LIN {X 0,Y 361.829,Z 158.416,A -85,B 0,C 180,E1 -12912.828,E2 -12912.828} C_VEL
LIN {X 0,Y 361.81,Z 158.413,A -85,B 0,C 180,E1 -12915.946,E2 -12915.946} C_VEL
LIN {X 0,Y 361.807,Z 158.415,A -85,B 0,C 180,E1 -12919.248,E2 -12919.248} C_VEL
LIN {X 0,Y 361.859,Z 158.41,A -85,B 0,C 180,E1 -12922.98,E2 -12922.98} C_VEL
LIN {X 0,Y 361.853,Z 158.414,A -85,B 0,C 180,E1 -12926.63,E2 -12926.63} C_VEL
LIN {X 0,Y 361.85,Z 158.408,A -85,B 0,C 180,E1 -12929.669,E2 -12929.669} C_VEL
LIN {X 0,Y 361.849,Z 158.408,A -85,B 0,C 180,E1 -12933.466,E2 -12933.466} C_VEL
LIN {X 0,Y 361.855,Z 158.408,A -85,B 0,C 180,E1 -12937.142,E2 -12937.142} C_VEL
LIN {X 0,Y 361.851,Z 158.41,A -85,B 0,C 180,E1 -12940.72,E2 -12940.72} C_VEL
LIN {X 0,Y 361.888,Z 158.409,A -85,B 0,C 180,E1 -12944.223,E2 -12944.223} C_VEL
LIN {X 0,Y 361.992,Z 158.393,A -85,B 0,C 180,E1 -12946.527,E2 -12946.527} C_VEL
LIN {X 0,Y 361.987,Z 158.395,A -85,B 0,C 180,E1 -12949.936,E2 -12949.936} C_VEL
LIN {X 0,Y 362.114,Z 158.375,A -85,B 0,C 180,E1 -12953.312,E2 -12953.312} C_VEL
LIN {X 0,Y 362.256,Z 158.361,A -85,B 0,C 180,E1 -12957.776,E2 -12957.776} C_VEL
LIN {X 0,Y 362.166,Z 158.369,A -85,B 0,C 180,E1 -12961.112,E2 -12961.112} C_VEL
LIN {X 0,Y 362.256,Z 158.36,A -85,B 0,C 180,E1 -12962.223,E2 -12962.223} C_VEL
LIN {X 0,Y 362.113,Z 158.375,A -85,B 0,C 180,E1 -12966.687,E2 -12966.687} C_VEL
LIN {X 0,Y 361.987,Z 158.394,A -85,B 0,C 180,E1 -12970.063,E2 -12970.063} C_VEL
LIN {X 0,Y 361.972,Z 158.397,A -85,B 0,C 180,E1 -12973.887,E2 -12973.887} C_VEL
LIN {X 0,Y 361.876,Z 158.406,A -85,B 0,C 180,E1 -12978.103,E2 -12978.103} C_VEL
LIN {X 0,Y 361.845,Z 158.413,A -85,B 0,C 180,E1 -12981.656,E2 -12981.656} C_VEL
LIN {X 0,Y 361.852,Z 158.413,A -85,B 0,C 180,E1 -12985.296,E2 -12985.296} C_VEL
LIN {X 0,Y 361.848,Z 158.412,A -85,B 0,C 180,E1 -12989.074,E2 -12989.074} C_VEL
LIN {X 0,Y 361.84,Z 158.412,A -85,B 0,C 180,E1 -12992.946,E2 -12992.946} C_VEL
LIN {X 0,Y 361.857,Z 158.409,A -85,B 0,C 180,E1 -12995.638,E2 -12995.638} C_VEL
LIN {X 0,Y 361.819,Z 158.417,A -85,B 0,C 180,E1 -12999.018,E2 -12999.018} C_VEL
LIN {X 0,Y 361.823,Z 158.415,A -85,B 0,C 180,E1 -13002.831,E2 -13002.831} C_VEL
LIN {X 0,Y 361.808,Z 158.413,A -85,B 0,C 180,E1 -13005.948,E2 -13005.948} C_VEL
LIN {X 0,Y 361.805,Z 158.416,A -85,B 0,C 180,E1 -13009.25,E2 -13009.25} C_VEL
LIN {X 0,Y 361.856,Z 158.412,A -85,B 0,C 180,E1 -13012.982,E2 -13012.982} C_VEL
LIN {X 0,Y 361.853,Z 158.412,A -85,B 0,C 180,E1 -13016.632,E2 -13016.632} C_VEL
LIN {X 0,Y 361.844,Z 158.411,A -85,B 0,C 180,E1 -13019.671,E2 -13019.671} C_VEL
LIN {X 0,Y 361.862,Z 158.495,A -85,B 0,C 180,E1 -13021.035,E2 -13021.035} C_VEL
LIN {X 0,Y 364.381,Z 171.266,A -85,B 0,C 180,E1 -13024.282,E2 -13024.282} C_VEL
LIN {X 0,Y 365.151,Z 176.441,A -85,B 0,C 180,E1 -13025.557,E2 -13025.557} C_VEL
LIN {X 0,Y 364.358,Z 186.129,A -85,B 0,C 180,E1 -13027.799,E2 -13027.799} C_VEL
LIN {X 0,Y 363.991,Z 190.26,A -85,B 0,C 180,E1 -13028.747,E2 -13028.747} C_VEL
LIN {X 0,Y 368.452,Z 222.561,A -85,B 0,C 180,E1 -13029.729,E2 -13029.729} C_VEL
LIN {X 0,Y 366.841,Z 299.767,A -85,B 0,C 180,E1 -13031.501,E2 -13031.501} C_VEL
LIN {X 0,Y 366.187,Z 313.467,A -85,B 0,C 180,E1 -13032.046,E2 -13032.046} C_VEL
LIN {X 0,Y 365.37,Z 326.351,A -85,B 0,C 180,E1 -13032.799,E2 -13032.799} C_VEL
LIN {X 0,Y 364.524,Z 338.673,A -85,B 0,C 180,E1 -13033.767,E2 -13033.767} C_VEL
LIN {X 0,Y 363.673,Z 349.679,A -85,B 0,C 180,E1 -13034.87,E2 -13034.87} C_VEL
LIN {X 0,Y 362.818,Z 360.759,A -85,B 0,C 180,E1 -13036.274,E2 -13036.274} C_VEL
LIN {X 0,Y 362.039,Z 369.703,A -85,B 0,C 180,E1 -13037.671,E2 -13037.671} C_VEL
LIN {X 0,Y 361.369,Z 377.07,A -85,B 0,C 180,E1 -13039.07,E2 -13039.07} C_VEL
LIN {X 0,Y 360.899,Z 384.28,A -85,B 0,C 180,E1 -13040.756,E2 -13040.756} C_VEL
LIN {X 0,Y 360.584,Z 390.846,A -85,B 0,C 180,E1 -13042.723,E2 -13042.723} C_VEL
LIN {X 0,Y 360.382,Z 395.127,A -85,B 0,C 180,E1 -13044.405,E2 -13044.405} C_VEL
LIN {X 0,Y 360.386,Z 397.376,A -85,B 0,C 180,E1 -13045.527,E2 -13045.527} C_VEL
LIN {X 0,Y 360.304,Z 399.111,A -85,B 0,C 180,E1 -13046.646,E2 -13046.646} C_VEL
LIN {X 0,Y 360.279,Z 400.423,A -85,B 0,C 180,E1 -13047.765,E2 -13047.765} C_VEL
LIN {X 0,Y 360.322,Z 401.322,A -85,B 0,C 180,E1 -13048.883,E2 -13048.883} C_VEL
LIN {X 0,Y 360.36,Z 401.765,A -85,B 0,C 180,E1 -13050.001,E2 -13050.001} C_VEL
LIN {X 0,Y 360.303,Z 401.777,A -85,B 0,C 180,E1 -13051.119,E2 -13051.119} C_VEL
LIN {X 0,Y 360.262,Z 401.385,A -85,B 0,C 180,E1 -13052.237,E2 -13052.237} C_VEL
LIN {X 0,Y 360.296,Z 400.589,A -85,B 0,C 180,E1 -13053.356,E2 -13053.356} C_VEL
LIN {X 0,Y 360.346,Z 399.333,A -85,B 0,C 180,E1 -13054.475,E2 -13054.475} C_VEL
LIN {X 0,Y 360.378,Z 397.037,A -85,B 0,C 180,E1 -13055.962,E2 -13055.962} C_VEL
LIN {X 0,Y 360.695,Z 392.947,A -85,B 0,C 180,E1 -13057.84,E2 -13057.84} C_VEL
LIN {X 0,Y 361.149,Z 388.099,A -85,B 0,C 180,E1 -13059.522,E2 -13059.522} C_VEL
LIN {X 0,Y 361.921,Z 380.826,A -85,B 0,C 180,E1 -13061.482,E2 -13061.482} C_VEL
LIN {X 0,Y 362.96,Z 372.947,A -85,B 0,C 180,E1 -13063.152,E2 -13063.152} C_VEL
LIN {X 0,Y 364.128,Z 363.132,A -85,B 0,C 180,E1 -13064.812,E2 -13064.812} C_VEL
LIN {X 0,Y 365.247,Z 353.009,A -85,B 0,C 180,E1 -13066.202,E2 -13066.202} C_VEL
LIN {X 0,Y 366.61,Z 341.672,A -85,B 0,C 180,E1 -13067.431,E2 -13067.431} C_VEL
LIN {X 0,Y 367.795,Z 330.68,A -85,B 0,C 180,E1 -13068.379,E2 -13068.379} C_VEL
LIN {X 0,Y 368.792,Z 318.696,A -85,B 0,C 180,E1 -13069.193,E2 -13069.193} C_VEL
LIN {X 0,Y 369.825,Z 305.614,A -85,B 0,C 180,E1 -13069.823,E2 -13069.823} C_VEL
LIN {X 0,Y 370.495,Z 292.075,A -85,B 0,C 180,E1 -13070.255,E2 -13070.255} C_VEL
LIN {X 0,Y 372.443,Z 222.981,A -85,B 0,C 180,E1 -13071.896,E2 -13071.896} C_VEL
LIN {X 0,Y 369.403,Z 203.708,A -85,B 0,C 180,E1 -13072.672,E2 -13072.672} C_VEL
LIN {X 0,Y 365.96,Z 188.136,A -85,B 0,C 180,E1 -13073.424,E2 -13073.424} C_VEL
LIN {X 0,Y 366.691,Z 181.612,A -85,B 0,C 180,E1 -13074.94,E2 -13074.94} C_VEL
LIN {X 0,Y 366.084,Z 176.728,A -85,B 0,C 180,E1 -13076.204,E2 -13076.204} C_VEL
LIN {X 0,Y 364.044,Z 167.054,A -85,B 0,C 180,E1 -13078.859,E2 -13078.859} C_VEL
LIN {X 0,Y 361.855,Z 158.412,A -85,B 0,C 180,E1 -13081.462,E2 -13081.462} C_VEL
LIN {X 0,Y 361.853,Z 158.411,A -85,B 0,C 180,E1 -13084.281,E2 -13084.281} C_VEL
LIN {X 0,Y 361.86,Z 158.409,A -85,B 0,C 180,E1 -13087.222,E2 -13087.222} C_VEL
LIN {X 0,Y 361.814,Z 158.417,A -85,B 0,C 180,E1 -13090.751,E2 -13090.751} C_VEL
LIN {X 0,Y 361.815,Z 158.413,A -85,B 0,C 180,E1 -13094.37,E2 -13094.37} C_VEL
LIN {X 0,Y 361.832,Z 158.409,A -85,B 0,C 180,E1 -13097.57,E2 -13097.57} C_VEL
LIN {X 0,Y 361.845,Z 158.405,A -85,B 0,C 180,E1 -13101.572,E2 -13101.572} C_VEL
LIN {X 0,Y 361.873,Z 158.407,A -85,B 0,C 180,E1 -13104.657,E2 -13104.657} C_VEL
LIN {X 0,Y 361.841,Z 158.413,A -85,B 0,C 180,E1 -13108.371,E2 -13108.371} C_VEL
LIN {X 0,Y 361.87,Z 158.406,A -85,B 0,C 180,E1 -13110.953,E2 -13110.953} C_VEL
LIN {X 0,Y 361.869,Z 158.405,A -85,B 0,C 180,E1 -13114.706,E2 -13114.706} C_VEL
LIN {X 0,Y 361.858,Z 158.41,A -85,B 0,C 180,E1 -13118.345,E2 -13118.345} C_VEL
LIN {X 0,Y 361.908,Z 158.403,A -85,B 0,C 180,E1 -13122.093,E2 -13122.093} C_VEL
LIN {X 0,Y 361.984,Z 158.394,A -85,B 0,C 180,E1 -13126.114,E2 -13126.114} C_VEL
LIN {X 0,Y 362.004,Z 158.394,A -85,B 0,C 180,E1 -13129.937,E2 -13129.937} C_VEL
LIN {X 0,Y 362.126,Z 158.38,A -85,B 0,C 180,E1 -13133.313,E2 -13133.313} C_VEL
LIN {X 0,Y 362.269,Z 158.361,A -85,B 0,C 180,E1 -13137.777,E2 -13137.777} C_VEL
LIN {X 0,Y 362.185,Z 158.387,A -85,B 0,C 180,E1 -13140.556,E2 -13140.556} C_VEL
LIN {X 0,Y 363.973,Z 165.762,A -85,B 0,C 180,E1 -13142.767,E2 -13142.767} C_VEL
LIN {X 0,Y 365.318,Z 172.142,A -85,B 0,C 180,E1 -13144.584,E2 -13144.584} C_VEL
LIN {X 0,Y 369.751,Z 182.829,A -85,B 0,C 180,E1 -13145.285,E2 -13145.285} C_VEL
LIN {X 0,Y 373.135,Z 198.483,A -85,B 0,C 180,E1 -13146,E2 -13146} C_VEL
LIN {X 0,Y 370.496,Z 280.618,A -85,B 0,C 180,E1 -13147.976,E2 -13147.976} C_VEL
LIN {X 0,Y 369.775,Z 293.95,A -85,B 0,C 180,E1 -13148.511,E2 -13148.511} C_VEL
LIN {X 0,Y 368.967,Z 305.625,A -85,B 0,C 180,E1 -13149.18,E2 -13149.18} C_VEL
LIN {X 0,Y 368.052,Z 316.889,A -85,B 0,C 180,E1 -13150.035,E2 -13150.035} C_VEL
LIN {X 0,Y 366.76,Z 329.226,A -85,B 0,C 180,E1 -13151.235,E2 -13151.235} C_VEL
LIN {X 0,Y 365.557,Z 339.475,A -85,B 0,C 180,E1 -13152.491,E2 -13152.491} C_VEL
LIN {X 0,Y 364.345,Z 349.032,A -85,B 0,C 180,E1 -13153.953,E2 -13153.953} C_VEL
LIN {X 0,Y 363.334,Z 357.164,A -85,B 0,C 180,E1 -13155.481,E2 -13155.481} C_VEL
LIN {X 0,Y 362.367,Z 364.439,A -85,B 0,C 180,E1 -13157.168,E2 -13157.168} C_VEL
LIN {X 0,Y 361.68,Z 369.722,A -85,B 0,C 180,E1 -13158.701,E2 -13158.701} C_VEL
LIN {X 0,Y 361.113,Z 374.595,A -85,B 0,C 180,E1 -13160.507,E2 -13160.507} C_VEL
LIN {X 0,Y 360.705,Z 378.217,A -85,B 0,C 180,E1 -13162.33,E2 -13162.33} C_VEL
LIN {X 0,Y 360.373,Z 380.677,A -85,B 0,C 180,E1 -13164.177,E2 -13164.177} C_VEL
LIN {X 0,Y 360.186,Z 382.039,A -85,B 0,C 180,E1 -13166.159,E2 -13166.159} C_VEL
LIN {X 0,Y 360.109,Z 381.931,A -85,B 0,C 180,E1 -13168.569,E2 -13168.569} C_VEL
LIN {X 0,Y 360.203,Z 380.066,A -85,B 0,C 180,E1 -13170.851,E2 -13170.851} C_VEL
LIN {X 0,Y 360.384,Z 377.741,A -85,B 0,C 180,E1 -13172.404,E2 -13172.404} C_VEL
LIN {X 0,Y 360.626,Z 373.429,A -85,B 0,C 180,E1 -13174.414,E2 -13174.414} C_VEL
LIN {X 0,Y 361.062,Z 367.492,A -85,B 0,C 180,E1 -13176.413,E2 -13176.413} C_VEL
LIN {X 0,Y 361.561,Z 361.004,A -85,B 0,C 180,E1 -13178.109,E2 -13178.109} C_VEL
LIN {X 0,Y 362.205,Z 352.769,A -85,B 0,C 180,E1 -13179.816,E2 -13179.816} C_VEL
LIN {X 0,Y 362.997,Z 343.553,A -85,B 0,C 180,E1 -13181.354,E2 -13181.354} C_VEL
LIN {X 0,Y 363.79,Z 333.043,A -85,B 0,C 180,E1 -13182.766,E2 -13182.766} C_VEL
LIN {X 0,Y 364.669,Z 322.16,A -85,B 0,C 180,E1 -13183.933,E2 -13183.933} C_VEL
LIN {X 0,Y 365.522,Z 310.748,A -85,B 0,C 180,E1 -13184.906,E2 -13184.906} C_VEL
LIN {X 0,Y 366.232,Z 298.142,A -85,B 0,C 180,E1 -13185.728,E2 -13185.728} C_VEL
LIN {X 0,Y 366.765,Z 284.578,A -85,B 0,C 180,E1 -13186.361,E2 -13186.361} C_VEL
LIN {X 0,Y 367.225,Z 270.752,A -85,B 0,C 180,E1 -13186.757,E2 -13186.757} C_VEL
LIN {X 0,Y 368.691,Z 195.693,A -85,B 0,C 180,E1 -13188.451,E2 -13188.451} C_VEL
LIN {X 0,Y 364.189,Z 170.992,A -85,B 0,C 180,E1 -13189.268,E2 -13189.268} C_VEL
LIN {X 0,Y 362.217,Z 160.038,A -85,B 0,C 180,E1 -13192.264,E2 -13192.264} C_VEL
LIN {X 0,Y 361.902,Z 158.407,A -85,B 0,C 180,E1 -13192.77,E2 -13192.77} C_VEL
LIN {X 0,Y 361.859,Z 158.407,A -85,B 0,C 180,E1 -13195.719,E2 -13195.719} C_VEL
LIN {X 0,Y 361.852,Z 158.408,A -85,B 0,C 180,E1 -13199.669,E2 -13199.669} C_VEL
LIN {X 0,Y 361.859,Z 158.407,A -85,B 0,C 180,E1 -13203.467,E2 -13203.467} C_VEL
LIN {X 0,Y 361.866,Z 158.406,A -85,B 0,C 180,E1 -13207.142,E2 -13207.142} C_VEL
LIN {X 0,Y 361.848,Z 158.41,A -85,B 0,C 180,E1 -13210.719,E2 -13210.719} C_VEL
LIN {X 0,Y 361.882,Z 158.404,A -85,B 0,C 180,E1 -13213.063,E2 -13213.063} C_VEL
LIN {X 0,Y 362.004,Z 158.391,A -85,B 0,C 180,E1 -13216.527,E2 -13216.527} C_VEL
LIN {X 0,Y 362,Z 158.395,A -85,B 0,C 180,E1 -13219.936,E2 -13219.936} C_VEL
LIN {X 0,Y 362.123,Z 158.375,A -85,B 0,C 180,E1 -13223.312,E2 -13223.312} C_VEL
LIN {X 0,Y 362.268,Z 158.361,A -85,B 0,C 180,E1 -13227.775,E2 -13227.775} C_VEL
LIN {X 0,Y 362.177,Z 158.368,A -85,B 0,C 180,E1 -13231.111,E2 -13231.111} C_VEL
LIN {X 0,Y 362.268,Z 158.358,A -85,B 0,C 180,E1 -13232.223,E2 -13232.223} C_VEL
LIN {X 0,Y 362.121,Z 158.374,A -85,B 0,C 180,E1 -13236.686,E2 -13236.686} C_VEL
LIN {X 0,Y 361.998,Z 158.391,A -85,B 0,C 180,E1 -13240.062,E2 -13240.062} C_VEL
LIN {X 0,Y 361.945,Z 158.395,A -85,B 0,C 180,E1 -13242.003,E2 -13242.003} C_VEL
LIN {X 0,Y 361.283,Z 158.481,A -85,B 0,C 180,E1 -13242.931,E2 -13242.931} C_VEL
LIN {X 0,Y 358.386,Z 158.839,A -85,B 0,C 180,E1 -13244.441,E2 -13244.441} C_VEL
LIN {X 0,Y 355.935,Z 159.149,A -85,B 0,C 180,E1 -13245.662,E2 -13245.662} C_VEL
LIN {X 0,Y 354.901,Z 159.274,A -85,B 0,C 180,E1 -13246.608,E2 -13246.608} C_VEL
LIN {X 0,Y 354.827,Z 159.284,A -85,B 0,C 180,E1 -13246.928,E2 -13246.928} C_VEL
LIN {X 0,Y 354.79,Z 159.291,A -85,B 0,C 180,E1 -13249.678,E2 -13249.678} C_VEL
LIN {X 0,Y 354.806,Z 159.286,A -85,B 0,C 180,E1 -13252.107,E2 -13252.107} C_VEL
LIN {X 0,Y 354.799,Z 159.287,A -85,B 0,C 180,E1 -13255.834,E2 -13255.834} C_VEL
LIN {X 0,Y 354.792,Z 159.289,A -85,B 0,C 180,E1 -13259.683,E2 -13259.683} C_VEL
LIN {X 0,Y 354.785,Z 159.288,A -85,B 0,C 180,E1 -13262.332,E2 -13262.332} C_VEL
LIN {X 0,Y 354.817,Z 159.285,A -85,B 0,C 180,E1 -13265.697,E2 -13265.697} C_VEL
LIN {X 0,Y 354.766,Z 159.293,A -85,B 0,C 180,E1 -13269.411,E2 -13269.411} C_VEL
LIN {X 0,Y 354.781,Z 159.294,A -85,B 0,C 180,E1 -13272.865,E2 -13272.865} C_VEL
LIN {X 0,Y 354.759,Z 159.292,A -85,B 0,C 180,E1 -13276.102,E2 -13276.102} C_VEL
LIN {X 0,Y 354.76,Z 159.294,A -85,B 0,C 180,E1 -13279.175,E2 -13279.175} C_VEL
LIN {X 0,Y 354.796,Z 159.29,A -85,B 0,C 180,E1 -13282.403,E2 -13282.403} C_VEL
LIN {X 0,Y 354.806,Z 159.289,A -85,B 0,C 180,E1 -13284.94,E2 -13284.94} C_VEL
LIN {X 0,Y 354.788,Z 159.292,A -85,B 0,C 180,E1 -13288.404,E2 -13288.404} C_VEL
LIN {X 0,Y 354.791,Z 159.287,A -85,B 0,C 180,E1 -13291.613,E2 -13291.613} C_VEL
LIN {X 0,Y 354.795,Z 159.287,A -85,B 0,C 180,E1 -13295.418,E2 -13295.418} C_VEL
LIN {X 0,Y 354.815,Z 159.285,A -85,B 0,C 180,E1 -13299.112,E2 -13299.112} C_VEL
LIN {X 0,Y 354.845,Z 159.283,A -85,B 0,C 180,E1 -13302.717,E2 -13302.717} C_VEL
LIN {X 0,Y 354.932,Z 159.276,A -85,B 0,C 180,E1 -13306.254,E2 -13306.254} C_VEL
LIN {X 0,Y 354.944,Z 159.27,A -85,B 0,C 180,E1 -13309.735,E2 -13309.735} C_VEL
LIN {X 0,Y 355.08,Z 159.251,A -85,B 0,C 180,E1 -13313.179,E2 -13313.179} C_VEL
LIN {X 0,Y 355.218,Z 159.238,A -85,B 0,C 180,E1 -13317.732,E2 -13317.732} C_VEL
LIN {X 0,Y 355.137,Z 159.244,A -85,B 0,C 180,E1 -13321.134,E2 -13321.134} C_VEL
LIN {X 0,Y 355.218,Z 159.237,A -85,B 0,C 180,E1 -13322.268,E2 -13322.268} C_VEL
LIN {X 0,Y 355.079,Z 159.251,A -85,B 0,C 180,E1 -13326.82,E2 -13326.82} C_VEL
LIN {X 0,Y 354.943,Z 159.27,A -85,B 0,C 180,E1 -13330.265,E2 -13330.265} C_VEL
LIN {X 0,Y 354.915,Z 159.274,A -85,B 0,C 180,E1 -13334.005,E2 -13334.005} C_VEL
LIN {X 0,Y 354.834,Z 159.284,A -85,B 0,C 180,E1 -13338.068,E2 -13338.068} C_VEL
LIN {X 0,Y 354.798,Z 159.287,A -85,B 0,C 180,E1 -13342.108,E2 -13342.108} C_VEL
LIN {X 0,Y 354.791,Z 159.289,A -85,B 0,C 180,E1 -13345.836,E2 -13345.836} C_VEL
LIN {X 0,Y 354.786,Z 159.291,A -85,B 0,C 180,E1 -13349.685,E2 -13349.685} C_VEL
LIN {X 0,Y 354.779,Z 159.289,A -85,B 0,C 180,E1 -13352.334,E2 -13352.334} C_VEL
LIN {X 0,Y 354.811,Z 159.286,A -85,B 0,C 180,E1 -13355.699,E2 -13355.699} C_VEL
LIN {X 0,Y 354.762,Z 159.294,A -85,B 0,C 180,E1 -13359.413,E2 -13359.413} C_VEL
LIN {X 0,Y 354.775,Z 159.294,A -85,B 0,C 180,E1 -13362.867,E2 -13362.867} C_VEL
LIN {X 0,Y 354.757,Z 159.292,A -85,B 0,C 180,E1 -13366.104,E2 -13366.104} C_VEL
LIN {X 0,Y 354.758,Z 159.295,A -85,B 0,C 180,E1 -13369.176,E2 -13369.176} C_VEL
LIN {X 0,Y 354.794,Z 159.289,A -85,B 0,C 180,E1 -13372.405,E2 -13372.405} C_VEL
LIN {X 0,Y 354.804,Z 159.29,A -85,B 0,C 180,E1 -13374.941,E2 -13374.941} C_VEL
LIN {X 0,Y 354.789,Z 159.29,A -85,B 0,C 180,E1 -13378.406,E2 -13378.406} C_VEL
LIN {X 0,Y 354.835,Z 159.397,A -85,B 0,C 180,E1 -13380.785,E2 -13380.785} C_VEL
LIN {X 0,Y 357.303,Z 171.951,A -85,B 0,C 180,E1 -13384.047,E2 -13384.047} C_VEL
LIN {X 0,Y 358.162,Z 177.252,A -85,B 0,C 180,E1 -13385.381,E2 -13385.381} C_VEL
LIN {X 0,Y 357.441,Z 186.368,A -85,B 0,C 180,E1 -13387.535,E2 -13387.535} C_VEL
LIN {X 0,Y 357.061,Z 190.013,A -85,B 0,C 180,E1 -13388.388,E2 -13388.388} C_VEL
LIN {X 0,Y 361.633,Z 222.954,A -85,B 0,C 180,E1 -13389.432,E2 -13389.432} C_VEL
LIN {X 0,Y 360.006,Z 298.965,A -85,B 0,C 180,E1 -13391.21,E2 -13391.21} C_VEL
LIN {X 0,Y 359.316,Z 312.831,A -85,B 0,C 180,E1 -13391.764,E2 -13391.764} C_VEL
LIN {X 0,Y 358.554,Z 324.868,A -85,B 0,C 180,E1 -13392.462,E2 -13392.462} C_VEL
LIN {X 0,Y 357.658,Z 337.442,A -85,B 0,C 180,E1 -13393.447,E2 -13393.447} C_VEL
LIN {X 0,Y 356.733,Z 348.739,A -85,B 0,C 180,E1 -13394.577,E2 -13394.577} C_VEL
LIN {X 0,Y 355.978,Z 358.93,A -85,B 0,C 180,E1 -13395.86,E2 -13395.86} C_VEL
LIN {X 0,Y 355.079,Z 368.978,A -85,B 0,C 180,E1 -13397.426,E2 -13397.426} C_VEL
LIN {X 0,Y 354.35,Z 376.436,A -85,B 0,C 180,E1 -13398.851,E2 -13398.851} C_VEL
LIN {X 0,Y 353.851,Z 383.761,A -85,B 0,C 180,E1 -13400.57,E2 -13400.57} C_VEL
LIN {X 0,Y 353.57,Z 388.695,A -85,B 0,C 180,E1 -13402.003,E2 -13402.003} C_VEL
LIN {X 0,Y 353.313,Z 394.163,A -85,B 0,C 180,E1 -13404.036,E2 -13404.036} C_VEL
LIN {X 0,Y 353.297,Z 397.027,A -85,B 0,C 180,E1 -13405.437,E2 -13405.437} C_VEL
LIN {X 0,Y 353.227,Z 398.801,A -85,B 0,C 180,E1 -13406.579,E2 -13406.579} C_VEL
LIN {X 0,Y 353.186,Z 400.136,A -85,B 0,C 180,E1 -13407.72,E2 -13407.72} C_VEL
LIN {X 0,Y 353.223,Z 401.059,A -85,B 0,C 180,E1 -13408.861,E2 -13408.861} C_VEL
LIN {X 0,Y 353.263,Z 401.552,A -85,B 0,C 180,E1 -13410.001,E2 -13410.001} C_VEL
LIN {X 0,Y 353.203,Z 401.589,A -85,B 0,C 180,E1 -13411.141,E2 -13411.141} C_VEL
LIN {X 0,Y 353.17,Z 401.223,A -85,B 0,C 180,E1 -13412.282,E2 -13412.282} C_VEL
LIN {X 0,Y 353.217,Z 400.456,A -85,B 0,C 180,E1 -13413.423,E2 -13413.423} C_VEL
LIN {X 0,Y 353.259,Z 399.246,A -85,B 0,C 180,E1 -13414.565,E2 -13414.565} C_VEL
LIN {X 0,Y 353.276,Z 397.264,A -85,B 0,C 180,E1 -13415.906,E2 -13415.906} C_VEL
LIN {X 0,Y 353.661,Z 392.957,A -85,B 0,C 180,E1 -13417.997,E2 -13417.997} C_VEL
LIN {X 0,Y 354.115,Z 388.159,A -85,B 0,C 180,E1 -13419.713,E2 -13419.713} C_VEL
LIN {X 0,Y 354.95,Z 380.941,A -85,B 0,C 180,E1 -13421.71,E2 -13421.71} C_VEL
LIN {X 0,Y 356.051,Z 373.182,A -85,B 0,C 180,E1 -13423.412,E2 -13423.412} C_VEL
LIN {X 0,Y 357.243,Z 363.769,A -85,B 0,C 180,E1 -13425.063,E2 -13425.063} C_VEL
LIN {X 0,Y 358.315,Z 354.591,A -85,B 0,C 180,E1 -13426.378,E2 -13426.378} C_VEL
LIN {X 0,Y 359.744,Z 343.77,A -85,B 0,C 180,E1 -13427.627,E2 -13427.627} C_VEL
LIN {X 0,Y 361.11,Z 331.597,A -85,B 0,C 180,E1 -13428.732,E2 -13428.732} C_VEL
LIN {X 0,Y 362.247,Z 318.821,A -85,B 0,C 180,E1 -13429.627,E2 -13429.627} C_VEL
LIN {X 0,Y 363.347,Z 305.934,A -85,B 0,C 180,E1 -13430.265,E2 -13430.265} C_VEL
LIN {X 0,Y 364.059,Z 291.534,A -85,B 0,C 180,E1 -13430.74,E2 -13430.74} C_VEL
LIN {X 0,Y 366.159,Z 223.616,A -85,B 0,C 180,E1 -13432.4,E2 -13432.4} C_VEL
LIN {X 0,Y 362.975,Z 203.973,A -85,B 0,C 180,E1 -13433.224,E2 -13433.224} C_VEL
LIN {X 0,Y 359.419,Z 187.839,A -85,B 0,C 180,E1 -13434.053,E2 -13434.053} C_VEL
LIN {X 0,Y 359.866,Z 182.107,A -85,B 0,C 180,E1 -13435.446,E2 -13435.446} C_VEL
LIN {X 0,Y 358.089,Z 172.427,A -85,B 0,C 180,E1 -13438.102,E2 -13438.102} C_VEL
LIN {X 0,Y 355.787,Z 162.976,A -85,B 0,C 180,E1 -13440.904,E2 -13440.904} C_VEL
LIN {X 0,Y 354.776,Z 159.295,A -85,B 0,C 180,E1 -13442.125,E2 -13442.125} C_VEL
LIN {X 0,Y 354.821,Z 159.286,A -85,B 0,C 180,E1 -13445.699,E2 -13445.699} C_VEL
LIN {X 0,Y 354.771,Z 159.295,A -85,B 0,C 180,E1 -13449.413,E2 -13449.413} C_VEL
LIN {X 0,Y 354.785,Z 159.29,A -85,B 0,C 180,E1 -13452.867,E2 -13452.867} C_VEL
LIN {X 0,Y 354.766,Z 159.286,A -85,B 0,C 180,E1 -13456.103,E2 -13456.103} C_VEL
LIN {X 0,Y 354.768,Z 159.287,A -85,B 0,C 180,E1 -13459.176,E2 -13459.176} C_VEL
LIN {X 0,Y 354.802,Z 159.287,A -85,B 0,C 180,E1 -13462.405,E2 -13462.405} C_VEL
LIN {X 0,Y 354.812,Z 159.29,A -85,B 0,C 180,E1 -13464.941,E2 -13464.941} C_VEL
LIN {X 0,Y 354.797,Z 159.289,A -85,B 0,C 180,E1 -13468.406,E2 -13468.406} C_VEL
LIN {X 0,Y 354.8,Z 159.285,A -85,B 0,C 180,E1 -13471.615,E2 -13471.615} C_VEL
LIN {X 0,Y 354.809,Z 159.286,A -85,B 0,C 180,E1 -13475.42,E2 -13475.42} C_VEL
LIN {X 0,Y 354.828,Z 159.28,A -85,B 0,C 180,E1 -13479.113,E2 -13479.113} C_VEL
LIN {X 0,Y 354.856,Z 159.283,A -85,B 0,C 180,E1 -13482.718,E2 -13482.718} C_VEL
LIN {X 0,Y 354.944,Z 159.271,A -85,B 0,C 180,E1 -13486.255,E2 -13486.255} C_VEL
LIN {X 0,Y 354.96,Z 159.272,A -85,B 0,C 180,E1 -13489.736,E2 -13489.736} C_VEL
LIN {X 0,Y 355.092,Z 159.256,A -85,B 0,C 180,E1 -13493.18,E2 -13493.18} C_VEL
LIN {X 0,Y 355.231,Z 159.237,A -85,B 0,C 180,E1 -13497.733,E2 -13497.733} C_VEL
LIN {X 0,Y 355.177,Z 159.338,A -85,B 0,C 180,E1 -13499.929,E2 -13499.929} C_VEL
LIN {X 0,Y 357.062,Z 166.798,A -85,B 0,C 180,E1 -13502.256,E2 -13502.256} C_VEL
LIN {X 0,Y 358.228,Z 172.673,A -85,B 0,C 180,E1 -13503.913,E2 -13503.913} C_VEL
LIN {X 0,Y 363.645,Z 184.715,A -85,B 0,C 180,E1 -13504.79,E2 -13504.79} C_VEL
LIN {X 0,Y 366.878,Z 199.629,A -85,B 0,C 180,E1 -13505.497,E2 -13505.497} C_VEL
LIN {X 0,Y 364.075,Z 281.33,A -85,B 0,C 180,E1 -13507.522,E2 -13507.522} C_VEL
LIN {X 0,Y 363.327,Z 294.218,A -85,B 0,C 180,E1 -13508.055,E2 -13508.055} C_VEL
LIN {X 0,Y 362.4,Z 306.756,A -85,B 0,C 180,E1 -13508.797,E2 -13508.797} C_VEL
LIN {X 0,Y 361.251,Z 319.341,A -85,B 0,C 180,E1 -13509.801,E2 -13509.801} C_VEL
LIN {X 0,Y 359.999,Z 330.799,A -85,B 0,C 180,E1 -13510.973,E2 -13510.973} C_VEL
LIN {X 0,Y 358.695,Z 340.853,A -85,B 0,C 180,E1 -13512.264,E2 -13512.264} C_VEL
LIN {X 0,Y 357.529,Z 349.603,A -85,B 0,C 180,E1 -13513.644,E2 -13513.644} C_VEL
LIN {X 0,Y 356.483,Z 357.482,A -85,B 0,C 180,E1 -13515.164,E2 -13515.164} C_VEL
LIN {X 0,Y 355.426,Z 364.981,A -85,B 0,C 180,E1 -13516.958,E2 -13516.958} C_VEL
LIN {X 0,Y 354.715,Z 370.084,A -85,B 0,C 180,E1 -13518.483,E2 -13518.483} C_VEL
LIN {X 0,Y 354.098,Z 374.921,A -85,B 0,C 180,E1 -13520.325,E2 -13520.325} C_VEL
LIN {X 0,Y 353.661,Z 378.511,A -85,B 0,C 180,E1 -13522.184,E2 -13522.184} C_VEL
LIN {X 0,Y 353.35,Z 380.682,A -85,B 0,C 180,E1 -13523.803,E2 -13523.803} C_VEL
LIN {X 0,Y 353.093,Z 382.221,A -85,B 0,C 180,E1 -13525.97,E2 -13525.97} C_VEL
LIN {X 0,Y 353.003,Z 382.453,A -85,B 0,C 180,E1 -13527.253,E2 -13527.253} C_VEL
LIN {X 0,Y 353.014,Z 381.969,A -85,B 0,C 180,E1 -13528.838,E2 -13528.838} C_VEL
LIN {X 0,Y 353.032,Z 381.26,A -85,B 0,C 180,E1 -13529.848,E2 -13529.848} C_VEL
LIN {X 0,Y 353.185,Z 378.877,A -85,B 0,C 180,E1 -13531.825,E2 -13531.825} C_VEL
LIN {X 0,Y 353.48,Z 375.079,A -85,B 0,C 180,E1 -13533.829,E2 -13533.829} C_VEL
LIN {X 0,Y 353.704,Z 370.93,A -85,B 0,C 180,E1 -13535.445,E2 -13535.445} C_VEL
LIN {X 0,Y 354.123,Z 365.839,A -85,B 0,C 180,E1 -13537.017,E2 -13537.017} C_VEL
LIN {X 0,Y 354.651,Z 359.392,A -85,B 0,C 180,E1 -13538.626,E2 -13538.626} C_VEL
LIN {X 0,Y 355.391,Z 350.69,A -85,B 0,C 180,E1 -13540.377,E2 -13540.377} C_VEL
LIN {X 0,Y 356.164,Z 341.093,A -85,B 0,C 180,E1 -13541.915,E2 -13541.915} C_VEL
LIN {X 0,Y 357.106,Z 330.02,A -85,B 0,C 180,E1 -13543.342,E2 -13543.342} C_VEL
LIN {X 0,Y 357.916,Z 319.863,A -85,B 0,C 180,E1 -13544.39,E2 -13544.39} C_VEL
LIN {X 0,Y 358.774,Z 308.064,A -85,B 0,C 180,E1 -13545.353,E2 -13545.353} C_VEL
LIN {X 0,Y 359.484,Z 295.268,A -85,B 0,C 180,E1 -13546.149,E2 -13546.149} C_VEL
LIN {X 0,Y 359.959,Z 282.978,A -85,B 0,C 180,E1 -13546.693,E2 -13546.693} C_VEL
LIN {X 0,Y 360.435,Z 265.632,A -85,B 0,C 180,E1 -13547.155,E2 -13547.155} C_VEL
LIN {X 0,Y 361.971,Z 196.986,A -85,B 0,C 180,E1 -13548.735,E2 -13548.735} C_VEL
LIN {X 0,Y 357.476,Z 172.71,A -85,B 0,C 180,E1 -13549.549,E2 -13549.549} C_VEL
LIN {X 0,Y 357.105,Z 171.169,A -85,B 0,C 180,E1 -13549.616,E2 -13549.616} C_VEL
LIN {X 0,Y 354.856,Z 159.284,A -85,B 0,C 180,E1 -13552.979,E2 -13552.979} C_VEL
LIN {X 0,Y 354.82,Z 159.288,A -85,B 0,C 180,E1 -13556.316,E2 -13556.316} C_VEL
LIN {X 0,Y 354.797,Z 159.288,A -85,B 0,C 180,E1 -13559,E2 -13559} C_VEL
LIN {X 0,Y 354.793,Z 159.287,A -85,B 0,C 180,E1 -13561.613,E2 -13561.613} C_VEL
LIN {X 0,Y 354.807,Z 159.285,A -85,B 0,C 180,E1 -13565.419,E2 -13565.419} C_VEL
LIN {X 0,Y 354.824,Z 159.283,A -85,B 0,C 180,E1 -13569.112,E2 -13569.112} C_VEL
LIN {X 0,Y 354.849,Z 159.281,A -85,B 0,C 180,E1 -13572.717,E2 -13572.717} C_VEL
LIN {X 0,Y 354.944,Z 159.273,A -85,B 0,C 180,E1 -13576.254,E2 -13576.254} C_VEL
LIN {X 0,Y 354.956,Z 159.27,A -85,B 0,C 180,E1 -13579.734,E2 -13579.734} C_VEL
LIN {X 0,Y 355.089,Z 159.25,A -85,B 0,C 180,E1 -13583.179,E2 -13583.179} C_VEL
LIN {X 0,Y 355.23,Z 159.238,A -85,B 0,C 180,E1 -13587.731,E2 -13587.731} C_VEL
LIN {X 0,Y 355.149,Z 159.243,A -85,B 0,C 180,E1 -13591.133,E2 -13591.133} C_VEL
LIN {X 0,Y 355.23,Z 159.234,A -85,B 0,C 180,E1 -13592.267,E2 -13592.267} C_VEL
LIN {X 0,Y 355.087,Z 159.251,A -85,B 0,C 180,E1 -13596.819,E2 -13596.819} C_VEL
LIN {X 0,Y 354.954,Z 159.268,A -85,B 0,C 180,E1 -13600.264,E2 -13600.264} C_VEL
LIN {X 0,Y 354.925,Z 159.272,A -85,B 0,C 180,E1 -13604.004,E2 -13604.004} C_VEL
LIN {X 0,Y 354.827,Z 159.284,A -85,B 0,C 180,E1 -13606.928,E2 -13606.928} C_VEL
LIN {X 0,Y 354.187,Z 159.369,A -85,B 0,C 180,E1 -13607.876,E2 -13607.876} C_VEL
LIN {X 0,Y 351.337,Z 159.727,A -85,B 0,C 180,E1 -13609.416,E2 -13609.416} C_VEL
LIN {X 0,Y 348.898,Z 160.028,A -85,B 0,C 180,E1 -13610.663,E2 -13610.663} C_VEL
LIN {X 0,Y 347.839,Z 160.157,A -85,B 0,C 180,E1 -13611.628,E2 -13611.628} C_VEL
LIN {X 0,Y 347.748,Z 160.166,A -85,B 0,C 180,E1 -13611.955,E2 -13611.955} C_VEL
LIN {X 0,Y 347.737,Z 160.17,A -85,B 0,C 180,E1 -13615.113,E2 -13615.113} C_VEL
LIN {X 0,Y 347.728,Z 160.169,A -85,B 0,C 180,E1 -13617.7,E2 -13617.7} C_VEL
LIN {X 0,Y 347.735,Z 160.166,A -85,B 0,C 180,E1 -13620.348,E2 -13620.348} C_VEL
LIN {X 0,Y 347.747,Z 160.165,A -85,B 0,C 180,E1 -13624.042,E2 -13624.042} C_VEL
LIN {X 0,Y 347.754,Z 160.167,A -85,B 0,C 180,E1 -13627.32,E2 -13627.32} C_VEL
LIN {X 0,Y 347.738,Z 160.167,A -85,B 0,C 180,E1 -13631.6,E2 -13631.6} C_VEL
LIN {X 0,Y 347.698,Z 160.175,A -85,B 0,C 180,E1 -13635.026,E2 -13635.026} C_VEL
LIN {X 0,Y 347.735,Z 160.168,A -85,B 0,C 180,E1 -13638.398,E2 -13638.398} C_VEL
LIN {X 0,Y 347.752,Z 160.17,A -85,B 0,C 180,E1 -13642.677,E2 -13642.677} C_VEL
LIN {X 0,Y 347.744,Z 160.166,A -85,B 0,C 180,E1 -13645.955,E2 -13645.955} C_VEL
LIN {X 0,Y 347.733,Z 160.167,A -85,B 0,C 180,E1 -13649.65,E2 -13649.65} C_VEL
LIN {X 0,Y 347.726,Z 160.167,A -85,B 0,C 180,E1 -13653.599,E2 -13653.599} C_VEL
LIN {X 0,Y 347.742,Z 160.169,A -85,B 0,C 180,E1 -13656.158,E2 -13656.158} C_VEL
LIN {X 0,Y 347.766,Z 160.164,A -85,B 0,C 180,E1 -13659.906,E2 -13659.906} C_VEL
LIN {X 0,Y 347.791,Z 160.16,A -85,B 0,C 180,E1 -13663.566,E2 -13663.566} C_VEL
LIN {X 0,Y 347.878,Z 160.148,A -85,B 0,C 180,E1 -13667.16,E2 -13667.16} C_VEL
LIN {X 0,Y 347.926,Z 160.144,A -85,B 0,C 180,E1 -13670.7,E2 -13670.7} C_VEL
LIN {X 0,Y 348.032,Z 160.134,A -85,B 0,C 180,E1 -13674.205,E2 -13674.205} C_VEL
LIN {X 0,Y 348.18,Z 160.114,A -85,B 0,C 180,E1 -13677.686,E2 -13677.686} C_VEL
LIN {X 0,Y 348.108,Z 160.12,A -85,B 0,C 180,E1 -13681.157,E2 -13681.157} C_VEL
LIN {X 0,Y 348.179,Z 160.113,A -85,B 0,C 180,E1 -13682.313,E2 -13682.313} C_VEL
LIN {X 0,Y 348.046,Z 160.128,A -85,B 0,C 180,E1 -13686.959,E2 -13686.959} C_VEL
LIN {X 0,Y 347.883,Z 160.148,A -85,B 0,C 180,E1 -13690.476,E2 -13690.476} C_VEL
LIN {X 0,Y 347.872,Z 160.151,A -85,B 0,C 180,E1 -13694.137,E2 -13694.137} C_VEL
LIN {X 0,Y 347.785,Z 160.161,A -85,B 0,C 180,E1 -13698.241,E2 -13698.241} C_VEL
LIN {X 0,Y 347.756,Z 160.168,A -85,B 0,C 180,E1 -13701.624,E2 -13701.624} C_VEL
LIN {X 0,Y 347.729,Z 160.17,A -85,B 0,C 180,E1 -13705.115,E2 -13705.115} C_VEL
LIN {X 0,Y 347.717,Z 160.171,A -85,B 0,C 180,E1 -13707.702,E2 -13707.702} C_VEL
LIN {X 0,Y 347.729,Z 160.167,A -85,B 0,C 180,E1 -13710.35,E2 -13710.35} C_VEL
LIN {X 0,Y 347.741,Z 160.166,A -85,B 0,C 180,E1 -13714.044,E2 -13714.044} C_VEL
LIN {X 0,Y 347.748,Z 160.169,A -85,B 0,C 180,E1 -13717.322,E2 -13717.322} C_VEL
LIN {X 0,Y 347.69,Z 160.172,A -85,B 0,C 180,E1 -13720.303,E2 -13720.303} C_VEL
LIN {X 0,Y 347.715,Z 160.171,A -85,B 0,C 180,E1 -13723.409,E2 -13723.409} C_VEL
LIN {X 0,Y 347.717,Z 160.172,A -85,B 0,C 180,E1 -13726.688,E2 -13726.688} C_VEL
LIN {X 0,Y 347.696,Z 160.172,A -85,B 0,C 180,E1 -13730.183,E2 -13730.183} C_VEL
LIN {X 0,Y 347.75,Z 160.169,A -85,B 0,C 180,E1 -13732.679,E2 -13732.679} C_VEL
LIN {X 0,Y 347.744,Z 160.165,A -85,B 0,C 180,E1 -13735.957,E2 -13735.957} C_VEL
LIN {X 0,Y 347.732,Z 160.169,A -85,B 0,C 180,E1 -13739.652,E2 -13739.652} C_VEL
LIN {X 0,Y 347.79,Z 160.347,A -85,B 0,C 180,E1 -13740.546,E2 -13740.546} C_VEL
LIN {X 0,Y 350.229,Z 172.617,A -85,B 0,C 180,E1 -13743.803,E2 -13743.803} C_VEL
LIN {X 0,Y 351.172,Z 179.103,A -85,B 0,C 180,E1 -13745.465,E2 -13745.465} C_VEL
LIN {X 0,Y 350.146,Z 189.908,A -85,B 0,C 180,E1 -13748.055,E2 -13748.055} C_VEL
LIN {X 0,Y 354.789,Z 224.029,A -85,B 0,C 180,E1 -13749.142,E2 -13749.142} C_VEL
LIN {X 0,Y 353.113,Z 298.775,A -85,B 0,C 180,E1 -13750.943,E2 -13750.943} C_VEL
LIN {X 0,Y 352.429,Z 312.609,A -85,B 0,C 180,E1 -13751.508,E2 -13751.508} C_VEL
LIN {X 0,Y 351.593,Z 325.132,A -85,B 0,C 180,E1 -13752.253,E2 -13752.253} C_VEL
LIN {X 0,Y 350.676,Z 337.608,A -85,B 0,C 180,E1 -13753.257,E2 -13753.257} C_VEL
LIN {X 0,Y 349.724,Z 348.831,A -85,B 0,C 180,E1 -13754.409,E2 -13754.409} C_VEL
LIN {X 0,Y 348.938,Z 359.21,A -85,B 0,C 180,E1 -13755.753,E2 -13755.753} C_VEL
LIN {X 0,Y 348.104,Z 368.149,A -85,B 0,C 180,E1 -13757.17,E2 -13757.17} C_VEL
LIN {X 0,Y 347.228,Z 377.097,A -85,B 0,C 180,E1 -13758.915,E2 -13758.915} C_VEL
LIN {X 0,Y 346.743,Z 384.218,A -85,B 0,C 180,E1 -13760.669,E2 -13760.669} C_VEL
LIN {X 0,Y 346.434,Z 389.893,A -85,B 0,C 180,E1 -13762.424,E2 -13762.424} C_VEL
LIN {X 0,Y 346.18,Z 395.072,A -85,B 0,C 180,E1 -13764.525,E2 -13764.525} C_VEL
LIN {X 0,Y 346.151,Z 398.471,A -85,B 0,C 180,E1 -13766.509,E2 -13766.509} C_VEL
LIN {X 0,Y 346.097,Z 399.836,A -85,B 0,C 180,E1 -13767.673,E2 -13767.673} C_VEL
LIN {X 0,Y 346.125,Z 400.789,A -85,B 0,C 180,E1 -13768.838,E2 -13768.838} C_VEL
LIN {X 0,Y 346.166,Z 401.327,A -85,B 0,C 180,E1 -13770.001,E2 -13770.001} C_VEL
LIN {X 0,Y 346.103,Z 401.401,A -85,B 0,C 180,E1 -13771.165,E2 -13771.165} C_VEL
LIN {X 0,Y 346.081,Z 401.061,A -85,B 0,C 180,E1 -13772.329,E2 -13772.329} C_VEL
LIN {X 0,Y 346.14,Z 400.319,A -85,B 0,C 180,E1 -13773.493,E2 -13773.493} C_VEL
LIN {X 0,Y 346.157,Z 399.157,A -85,B 0,C 180,E1 -13774.659,E2 -13774.659} C_VEL
LIN {X 0,Y 346.197,Z 397.43,A -85,B 0,C 180,E1 -13775.886,E2 -13775.886} C_VEL
LIN {X 0,Y 346.479,Z 394.263,A -85,B 0,C 180,E1 -13777.577,E2 -13777.577} C_VEL
LIN {X 0,Y 346.914,Z 389.928,A -85,B 0,C 180,E1 -13779.328,E2 -13779.328} C_VEL
LIN {X 0,Y 347.727,Z 383.357,A -85,B 0,C 180,E1 -13781.366,E2 -13781.366} C_VEL
LIN {X 0,Y 348.717,Z 376.212,A -85,B 0,C 180,E1 -13783.106,E2 -13783.106} C_VEL
LIN {X 0,Y 350.023,Z 367.289,A -85,B 0,C 180,E1 -13784.834,E2 -13784.834} C_VEL
LIN {X 0,Y 351.101,Z 358.202,A -85,B 0,C 180,E1 -13786.275,E2 -13786.275} C_VEL
LIN {X 0,Y 352.494,Z 348.25,A -85,B 0,C 180,E1 -13787.552,E2 -13787.552} C_VEL
LIN {X 0,Y 353.916,Z 337.352,A -85,B 0,C 180,E1 -13788.676,E2 -13788.676} C_VEL
LIN {X 0,Y 355.199,Z 325.372,A -85,B 0,C 180,E1 -13789.656,E2 -13789.656} C_VEL
LIN {X 0,Y 356.32,Z 313.118,A -85,B 0,C 180,E1 -13790.419,E2 -13790.419} C_VEL
LIN {X 0,Y 357.401,Z 299.581,A -85,B 0,C 180,E1 -13790.994,E2 -13790.994} C_VEL
LIN {X 0,Y 358.147,Z 278.846,A -85,B 0,C 180,E1 -13791.552,E2 -13791.552} C_VEL
LIN {X 0,Y 359.858,Z 224.384,A -85,B 0,C 180,E1 -13792.925,E2 -13792.925} C_VEL
LIN {X 0,Y 356.793,Z 205.328,A -85,B 0,C 180,E1 -13793.762,E2 -13793.762} C_VEL
LIN {X 0,Y 352.865,Z 187.637,A -85,B 0,C 180,E1 -13794.701,E2 -13794.701} C_VEL
LIN {X 0,Y 353.067,Z 183.832,A -85,B 0,C 180,E1 -13795.656,E2 -13795.656} C_VEL
LIN {X 0,Y 351.327,Z 174.362,A -85,B 0,C 180,E1 -13798.336,E2 -13798.336} C_VEL
LIN {X 0,Y 349.364,Z 166.05,A -85,B 0,C 180,E1 -13800.862,E2 -13800.862} C_VEL
LIN {X 0,Y 347.741,Z 160.171,A -85,B 0,C 180,E1 -13802.84,E2 -13802.84} C_VEL
LIN {X 0,Y 347.769,Z 160.165,A -85,B 0,C 180,E1 -13806.065,E2 -13806.065} C_VEL
LIN {X 0,Y 347.733,Z 160.172,A -85,B 0,C 180,E1 -13808.796,E2 -13808.796} C_VEL
LIN {X 0,Y 347.744,Z 160.166,A -85,B 0,C 180,E1 -13811.832,E2 -13811.832} C_VEL
LIN {X 0,Y 347.704,Z 160.17,A -85,B 0,C 180,E1 -13815.028,E2 -13815.028} C_VEL
LIN {X 0,Y 347.744,Z 160.162,A -85,B 0,C 180,E1 -13818.4,E2 -13818.4} C_VEL
LIN {X 0,Y 347.758,Z 160.167,A -85,B 0,C 180,E1 -13822.679,E2 -13822.679} C_VEL
LIN {X 0,Y 347.752,Z 160.167,A -85,B 0,C 180,E1 -13825.957,E2 -13825.957} C_VEL
LIN {X 0,Y 347.742,Z 160.164,A -85,B 0,C 180,E1 -13829.651,E2 -13829.651} C_VEL
LIN {X 0,Y 347.739,Z 160.167,A -85,B 0,C 180,E1 -13833.6,E2 -13833.6} C_VEL
LIN {X 0,Y 347.752,Z 160.165,A -85,B 0,C 180,E1 -13836.159,E2 -13836.159} C_VEL
LIN {X 0,Y 347.782,Z 160.16,A -85,B 0,C 180,E1 -13839.908,E2 -13839.908} C_VEL
LIN {X 0,Y 347.802,Z 160.161,A -85,B 0,C 180,E1 -13843.567,E2 -13843.567} C_VEL
LIN {X 0,Y 347.891,Z 160.152,A -85,B 0,C 180,E1 -13847.161,E2 -13847.161} C_VEL
LIN {X 0,Y 347.939,Z 160.148,A -85,B 0,C 180,E1 -13850.701,E2 -13850.701} C_VEL
LIN {X 0,Y 348.044,Z 160.135,A -85,B 0,C 180,E1 -13854.206,E2 -13854.206} C_VEL
LIN {X 0,Y 348.193,Z 160.114,A -85,B 0,C 180,E1 -13857.687,E2 -13857.687} C_VEL
LIN {X 0,Y 348.136,Z 160.187,A -85,B 0,C 180,E1 -13859.205,E2 -13859.205} C_VEL
LIN {X 0,Y 350.146,Z 167.92,A -85,B 0,C 180,E1 -13861.726,E2 -13861.726} C_VEL
LIN {X 0,Y 351.133,Z 172.852,A -85,B 0,C 180,E1 -13863.192,E2 -13863.192} C_VEL
LIN {X 0,Y 357.453,Z 186.69,A -85,B 0,C 180,E1 -13864.253,E2 -13864.253} C_VEL
LIN {X 0,Y 360.244,Z 198.517,A -85,B 0,C 180,E1 -13864.873,E2 -13864.873} C_VEL
LIN {X 0,Y 360.685,Z 201.779,A -85,B 0,C 180,E1 -13865.008,E2 -13865.008} C_VEL
LIN {X 0,Y 357.722,Z 281.473,A -85,B 0,C 180,E1 -13867.018,E2 -13867.018} C_VEL
LIN {X 0,Y 356.926,Z 294.523,A -85,B 0,C 180,E1 -13867.567,E2 -13867.567} C_VEL
LIN {X 0,Y 356.014,Z 306.442,A -85,B 0,C 180,E1 -13868.282,E2 -13868.282} C_VEL
LIN {X 0,Y 354.859,Z 318.603,A -85,B 0,C 180,E1 -13869.26,E2 -13869.26} C_VEL
LIN {X 0,Y 353.457,Z 330.261,A -85,B 0,C 180,E1 -13870.454,E2 -13870.454} C_VEL
LIN {X 0,Y 352.151,Z 340.379,A -85,B 0,C 180,E1 -13871.76,E2 -13871.76} C_VEL
LIN {X 0,Y 350.73,Z 350.169,A -85,B 0,C 180,E1 -13873.323,E2 -13873.323} C_VEL
LIN {X 0,Y 349.552,Z 358.464,A -85,B 0,C 180,E1 -13874.971,E2 -13874.971} C_VEL
LIN {X 0,Y 348.501,Z 365.435,A -85,B 0,C 180,E1 -13876.701,E2 -13876.701} C_VEL
LIN {X 0,Y 347.75,Z 370.389,A -85,B 0,C 180,E1 -13878.217,E2 -13878.217} C_VEL
LIN {X 0,Y 347.072,Z 375.276,A -85,B 0,C 180,E1 -13880.136,E2 -13880.136} C_VEL
LIN {X 0,Y 346.747,Z 377.771,A -85,B 0,C 180,E1 -13881.398,E2 -13881.398} C_VEL
LIN {X 0,Y 346.478,Z 379.752,A -85,B 0,C 180,E1 -13882.669,E2 -13882.669} C_VEL
LIN {X 0,Y 346.238,Z 381.264,A -85,B 0,C 180,E1 -13884.016,E2 -13884.016} C_VEL
LIN {X 0,Y 346.075,Z 382.184,A -85,B 0,C 180,E1 -13885.244,E2 -13885.244} C_VEL
LIN {X 0,Y 345.967,Z 382.614,A -85,B 0,C 180,E1 -13886.641,E2 -13886.641} C_VEL
LIN {X 0,Y 345.905,Z 382.534,A -85,B 0,C 180,E1 -13887.86,E2 -13887.86} C_VEL
LIN {X 0,Y 345.935,Z 381.91,A -85,B 0,C 180,E1 -13889.182,E2 -13889.182} C_VEL
LIN {X 0,Y 346.073,Z 379.555,A -85,B 0,C 180,E1 -13891.467,E2 -13891.467} C_VEL
LIN {X 0,Y 346.32,Z 376.583,A -85,B 0,C 180,E1 -13893.225,E2 -13893.225} C_VEL
LIN {X 0,Y 346.575,Z 371.927,A -85,B 0,C 180,E1 -13895.211,E2 -13895.211} C_VEL
LIN {X 0,Y 347.05,Z 366.199,A -85,B 0,C 180,E1 -13897.047,E2 -13897.047} C_VEL
LIN {X 0,Y 347.618,Z 359.246,A -85,B 0,C 180,E1 -13898.811,E2 -13898.811} C_VEL
LIN {X 0,Y 348.399,Z 350.509,A -85,B 0,C 180,E1 -13900.584,E2 -13900.584} C_VEL
LIN {X 0,Y 349.138,Z 341.479,A -85,B 0,C 180,E1 -13902.056,E2 -13902.056} C_VEL
LIN {X 0,Y 350.019,Z 331.157,A -85,B 0,C 180,E1 -13903.425,E2 -13903.425} C_VEL
LIN {X 0,Y 350.869,Z 321.033,A -85,B 0,C 180,E1 -13904.513,E2 -13904.513} C_VEL
LIN {X 0,Y 351.733,Z 310.455,A -85,B 0,C 180,E1 -13905.426,E2 -13905.426} C_VEL
LIN {X 0,Y 352.466,Z 297.467,A -85,B 0,C 180,E1 -13906.288,E2 -13906.288} C_VEL
LIN {X 0,Y 352.986,Z 284.672,A -85,B 0,C 180,E1 -13906.899,E2 -13906.899} C_VEL
LIN {X 0,Y 353.469,Z 270.73,A -85,B 0,C 180,E1 -13907.312,E2 -13907.312} C_VEL
LIN {X 0,Y 355.172,Z 198.097,A -85,B 0,C 180,E1 -13909.03,E2 -13909.03} C_VEL
LIN {X 0,Y 350.932,Z 174.872,A -85,B 0,C 180,E1 -13909.824,E2 -13909.824} C_VEL
LIN {X 0,Y 349.921,Z 171.251,A -85,B 0,C 180,E1 -13910.005,E2 -13910.005} C_VEL
LIN {X 0,Y 347.82,Z 160.161,A -85,B 0,C 180,E1 -13913.196,E2 -13913.196} C_VEL
LIN {X 0,Y 347.738,Z 160.168,A -85,B 0,C 180,E1 -13916.927,E2 -13916.927} C_VEL
LIN {X 0,Y 347.754,Z 160.169,A -85,B 0,C 180,E1 -13920.346,E2 -13920.346} C_VEL
LIN {X 0,Y 347.737,Z 160.166,A -85,B 0,C 180,E1 -13923.599,E2 -13923.599} C_VEL
LIN {X 0,Y 347.753,Z 160.169,A -85,B 0,C 180,E1 -13926.158,E2 -13926.158} C_VEL
LIN {X 0,Y 347.771,Z 160.165,A -85,B 0,C 180,E1 -13929.906,E2 -13929.906} C_VEL
LIN {X 0,Y 347.795,Z 160.16,A -85,B 0,C 180,E1 -13933.566,E2 -13933.566} C_VEL
LIN {X 0,Y 347.89,Z 160.147,A -85,B 0,C 180,E1 -13937.16,E2 -13937.16} C_VEL
LIN {X 0,Y 347.938,Z 160.141,A -85,B 0,C 180,E1 -13940.7,E2 -13940.7} C_VEL
LIN {X 0,Y 348.041,Z 160.132,A -85,B 0,C 180,E1 -13944.204,E2 -13944.204} C_VEL
LIN {X 0,Y 348.191,Z 160.114,A -85,B 0,C 180,E1 -13947.685,E2 -13947.685} C_VEL
LIN {X 0,Y 348.12,Z 160.119,A -85,B 0,C 180,E1 -13951.156,E2 -13951.156} C_VEL
LIN {X 0,Y 348.191,Z 160.111,A -85,B 0,C 180,E1 -13952.313,E2 -13952.313} C_VEL
LIN {X 0,Y 348.055,Z 160.127,A -85,B 0,C 180,E1 -13956.958,E2 -13956.958} C_VEL
LIN {X 0,Y 347.894,Z 160.147,A -85,B 0,C 180,E1 -13960.474,E2 -13960.474} C_VEL
LIN {X 0,Y 347.882,Z 160.149,A -85,B 0,C 180,E1 -13964.136,E2 -13964.136} C_VEL
LIN {X 0,Y 347.794,Z 160.159,A -85,B 0,C 180,E1 -13968.239,E2 -13968.239} C_VEL
LIN {X 0,Y 347.748,Z 160.166,A -85,B 0,C 180,E1 -13971.955,E2 -13971.955} C_VEL
LIN {X 0,Y 347.076,Z 160.252,A -85,B 0,C 180,E1 -13972.921,E2 -13972.921} C_VEL
LIN {X 0,Y 344.253,Z 160.601,A -85,B 0,C 180,E1 -13974.494,E2 -13974.494} C_VEL
LIN {X 0,Y 341.853,Z 160.903,A -85,B 0,C 180,E1 -13975.767,E2 -13975.767} C_VEL
LIN {X 0,Y 340.801,Z 161.034,A -85,B 0,C 180,E1 -13976.752,E2 -13976.752} C_VEL
LIN {X 0,Y 340.704,Z 161.045,A -85,B 0,C 180,E1 -13977.085,E2 -13977.085} C_VEL
LIN {X 0,Y 340.691,Z 161.049,A -85,B 0,C 180,E1 -13981.044,E2 -13981.044} C_VEL
LIN {X 0,Y 340.714,Z 161.045,A -85,B 0,C 180,E1 -13985.278,E2 -13985.278} C_VEL
LIN {X 0,Y 340.691,Z 161.045,A -85,B 0,C 180,E1 -13988.381,E2 -13988.381} C_VEL
LIN {X 0,Y 340.69,Z 161.044,A -85,B 0,C 180,E1 -13992.043,E2 -13992.043} C_VEL
LIN {X 0,Y 340.646,Z 161.05,A -85,B 0,C 180,E1 -13996.226,E2 -13996.226} C_VEL
LIN {X 0,Y 340.666,Z 161.052,A -85,B 0,C 180,E1 -13998.687,E2 -13998.687} C_VEL
LIN {X 0,Y 340.714,Z 161.041,A -85,B 0,C 180,E1 -14001.77,E2 -14001.77} C_VEL
LIN {X 0,Y 340.718,Z 161.04,A -85,B 0,C 180,E1 -14005.594,E2 -14005.594} C_VEL
LIN {X 0,Y 340.688,Z 161.047,A -85,B 0,C 180,E1 -14008.954,E2 -14008.954} C_VEL
LIN {X 0,Y 340.704,Z 161.044,A -85,B 0,C 180,E1 -14013.011,E2 -14013.011} C_VEL
LIN {X 0,Y 340.694,Z 161.045,A -85,B 0,C 180,E1 -14016.924,E2 -14016.924} C_VEL
LIN {X 0,Y 340.699,Z 161.045,A -85,B 0,C 180,E1 -14020.728,E2 -14020.728} C_VEL
LIN {X 0,Y 340.786,Z 161.036,A -85,B 0,C 180,E1 -14024.449,E2 -14024.449} C_VEL
LIN {X 0,Y 340.838,Z 161.031,A -85,B 0,C 180,E1 -14028.1,E2 -14028.1} C_VEL
LIN {X 0,Y 340.973,Z 161.011,A -85,B 0,C 180,E1 -14031.704,E2 -14031.704} C_VEL
LIN {X 0,Y 341.007,Z 161.01,A -85,B 0,C 180,E1 -14034.085,E2 -14034.085} C_VEL
LIN {X 0,Y 341.117,Z 160.993,A -85,B 0,C 180,E1 -14037.638,E2 -14037.638} C_VEL
LIN {X 0,Y 341.08,Z 160.996,A -85,B 0,C 180,E1 -14041.18,E2 -14041.18} C_VEL
LIN {X 0,Y 341.116,Z 160.992,A -85,B 0,C 180,E1 -14042.361,E2 -14042.361} C_VEL
LIN {X 0,Y 341.006,Z 161.01,A -85,B 0,C 180,E1 -14045.914,E2 -14045.914} C_VEL
LIN {X 0,Y 340.956,Z 161.012,A -85,B 0,C 180,E1 -14048.356,E2 -14048.356} C_VEL
LIN {X 0,Y 340.837,Z 161.029,A -85,B 0,C 180,E1 -14051.899,E2 -14051.899} C_VEL
LIN {X 0,Y 340.781,Z 161.038,A -85,B 0,C 180,E1 -14055.551,E2 -14055.551} C_VEL
LIN {X 0,Y 340.684,Z 161.048,A -85,B 0,C 180,E1 -14059.273,E2 -14059.273} C_VEL
LIN {X 0,Y 340.692,Z 161.046,A -85,B 0,C 180,E1 -14063.075,E2 -14063.075} C_VEL
LIN {X 0,Y 340.702,Z 161.045,A -85,B 0,C 180,E1 -14066.989,E2 -14066.989} C_VEL
LIN {X 0,Y 340.685,Z 161.048,A -85,B 0,C 180,E1 -14071.046,E2 -14071.046} C_VEL
LIN {X 0,Y 340.709,Z 161.047,A -85,B 0,C 180,E1 -14075.28,E2 -14075.28} C_VEL
LIN {X 0,Y 340.686,Z 161.045,A -85,B 0,C 180,E1 -14078.383,E2 -14078.383} C_VEL
LIN {X 0,Y 340.684,Z 161.045,A -85,B 0,C 180,E1 -14082.044,E2 -14082.044} C_VEL
LIN {X 0,Y 340.644,Z 161.05,A -85,B 0,C 180,E1 -14086.228,E2 -14086.228} C_VEL
LIN {X 0,Y 340.663,Z 161.051,A -85,B 0,C 180,E1 -14088.689,E2 -14088.689} C_VEL
LIN {X 0,Y 340.713,Z 161.041,A -85,B 0,C 180,E1 -14091.772,E2 -14091.772} C_VEL
LIN {X 0,Y 340.718,Z 161.041,A -85,B 0,C 180,E1 -14095.597,E2 -14095.597} C_VEL
LIN {X 0,Y 340.688,Z 161.048,A -85,B 0,C 180,E1 -14098.956,E2 -14098.956} C_VEL
LIN {X 0,Y 340.697,Z 161.065,A -85,B 0,C 180,E1 -14100.24,E2 -14100.24} C_VEL
LIN {X 0,Y 343.118,Z 173.12,A -85,B 0,C 180,E1 -14103.513,E2 -14103.513} C_VEL
LIN {X 0,Y 344.17,Z 179.767,A -85,B 0,C 180,E1 -14105.254,E2 -14105.254} C_VEL
LIN {X 0,Y 343.51,Z 187.384,A -85,B 0,C 180,E1 -14107.126,E2 -14107.126} C_VEL
LIN {X 0,Y 343.238,Z 189.75,A -85,B 0,C 180,E1 -14107.702,E2 -14107.702} C_VEL
LIN {X 0,Y 347.969,Z 224.515,A -85,B 0,C 180,E1 -14108.842,E2 -14108.842} C_VEL
LIN {X 0,Y 346.221,Z 298.493,A -85,B 0,C 180,E1 -14110.664,E2 -14110.664} C_VEL
LIN {X 0,Y 345.525,Z 312.332,A -85,B 0,C 180,E1 -14111.24,E2 -14111.24} C_VEL
LIN {X 0,Y 344.636,Z 325.371,A -85,B 0,C 180,E1 -14112.036,E2 -14112.036} C_VEL
LIN {X 0,Y 343.698,Z 337.762,A -85,B 0,C 180,E1 -14113.06,E2 -14113.06} C_VEL
LIN {X 0,Y 342.719,Z 348.914,A -85,B 0,C 180,E1 -14114.235,E2 -14114.235} C_VEL
LIN {X 0,Y 341.822,Z 359.991,A -85,B 0,C 180,E1 -14115.717,E2 -14115.717} C_VEL
LIN {X 0,Y 340.968,Z 368.98,A -85,B 0,C 180,E1 -14117.199,E2 -14117.199} C_VEL
LIN {X 0,Y 340.226,Z 376.383,A -85,B 0,C 180,E1 -14118.684,E2 -14118.684} C_VEL
LIN {X 0,Y 339.709,Z 383.634,A -85,B 0,C 180,E1 -14120.474,E2 -14120.474} C_VEL
LIN {X 0,Y 339.369,Z 389.39,A -85,B 0,C 180,E1 -14122.265,E2 -14122.265} C_VEL
LIN {X 0,Y 339.129,Z 394.021,A -85,B 0,C 180,E1 -14124.12,E2 -14124.12} C_VEL
LIN {X 0,Y 339.105,Z 396.24,A -85,B 0,C 180,E1 -14125.246,E2 -14125.246} C_VEL
LIN {X 0,Y 339.077,Z 398.138,A -85,B 0,C 180,E1 -14126.436,E2 -14126.436} C_VEL
LIN {X 0,Y 339.011,Z 399.537,A -85,B 0,C 180,E1 -14127.625,E2 -14127.625} C_VEL
LIN {X 0,Y 339.027,Z 400.518,A -85,B 0,C 180,E1 -14128.813,E2 -14128.813} C_VEL
LIN {X 0,Y 339.07,Z 401.09,A -85,B 0,C 180,E1 -14130.001,E2 -14130.001} C_VEL
LIN {X 0,Y 339.006,Z 401.214,A -85,B 0,C 180,E1 -14131.189,E2 -14131.189} C_VEL
LIN {X 0,Y 338.996,Z 400.899,A -85,B 0,C 180,E1 -14132.377,E2 -14132.377} C_VEL
LIN {X 0,Y 339.064,Z 400.185,A -85,B 0,C 180,E1 -14133.566,E2 -14133.566} C_VEL
LIN {X 0,Y 339.06,Z 399.064,A -85,B 0,C 180,E1 -14134.757,E2 -14134.757} C_VEL
LIN {X 0,Y 339.197,Z 396.539,A -85,B 0,C 180,E1 -14136.544,E2 -14136.544} C_VEL
LIN {X 0,Y 339.567,Z 392.992,A -85,B 0,C 180,E1 -14138.331,E2 -14138.331} C_VEL
LIN {X 0,Y 340.082,Z 388.342,A -85,B 0,C 180,E1 -14140.118,E2 -14140.118} C_VEL
LIN {X 0,Y 340.846,Z 382.46,A -85,B 0,C 180,E1 -14141.9,E2 -14141.9} C_VEL
LIN {X 0,Y 342.053,Z 375.093,A -85,B 0,C 180,E1 -14143.668,E2 -14143.668} C_VEL
LIN {X 0,Y 343.404,Z 365.995,A -85,B 0,C 180,E1 -14145.431,E2 -14145.431} C_VEL
LIN {X 0,Y 344.643,Z 356.74,A -85,B 0,C 180,E1 -14146.894,E2 -14146.894} C_VEL
LIN {X 0,Y 346.149,Z 346.498,A -85,B 0,C 180,E1 -14148.191,E2 -14148.191} C_VEL
LIN {X 0,Y 347.648,Z 335.262,A -85,B 0,C 180,E1 -14149.333,E2 -14149.333} C_VEL
LIN {X 0,Y 349.016,Z 322.8,A -85,B 0,C 180,E1 -14150.327,E2 -14150.327} C_VEL
LIN {X 0,Y 350.172,Z 310.256,A -85,B 0,C 180,E1 -14151.063,E2 -14151.063} C_VEL
LIN {X 0,Y 351.194,Z 296.61,A -85,B 0,C 180,E1 -14151.614,E2 -14151.614} C_VEL
LIN {X 0,Y 353.69,Z 225.636,A -85,B 0,C 180,E1 -14153.456,E2 -14153.456} C_VEL
LIN {X 0,Y 350.917,Z 207.783,A -85,B 0,C 180,E1 -14154.266,E2 -14154.266} C_VEL
LIN {X 0,Y 346.766,Z 189.442,A -85,B 0,C 180,E1 -14155.268,E2 -14155.268} C_VEL
LIN {X 0,Y 346.324,Z 187.431,A -85,B 0,C 180,E1 -14155.385,E2 -14155.385} C_VEL
LIN {X 0,Y 345.889,Z 182.983,A -85,B 0,C 180,E1 -14156.617,E2 -14156.617} C_VEL
LIN {X 0,Y 343.82,Z 172.718,A -85,B 0,C 180,E1 -14159.677,E2 -14159.677} C_VEL
LIN {X 0,Y 341.512,Z 164.203,A -85,B 0,C 180,E1 -14162.462,E2 -14162.462} C_VEL
LIN {X 0,Y 340.703,Z 161.047,A -85,B 0,C 180,E1 -14163.58,E2 -14163.58} C_VEL
LIN {X 0,Y 340.703,Z 161.048,A -85,B 0,C 180,E1 -14166.743,E2 -14166.743} C_VEL
LIN {X 0,Y 340.654,Z 161.051,A -85,B 0,C 180,E1 -14170.24,E2 -14170.24} C_VEL
LIN {X 0,Y 340.675,Z 161.048,A -85,B 0,C 180,E1 -14172.906,E2 -14172.906} C_VEL
LIN {X 0,Y 340.676,Z 161.042,A -85,B 0,C 180,E1 -14177.096,E2 -14177.096} C_VEL
LIN {X 0,Y 340.658,Z 161.048,A -85,B 0,C 180,E1 -14180.242,E2 -14180.242} C_VEL
LIN {X 0,Y 340.71,Z 161.04,A -85,B 0,C 180,E1 -14183.561,E2 -14183.561} C_VEL
LIN {X 0,Y 340.695,Z 161.044,A -85,B 0,C 180,E1 -14186.154,E2 -14186.154} C_VEL
LIN {X 0,Y 340.725,Z 161.04,A -85,B 0,C 180,E1 -14190.035,E2 -14190.035} C_VEL
LIN {X 0,Y 340.714,Z 161.042,A -85,B 0,C 180,E1 -14193.012,E2 -14193.012} C_VEL
LIN {X 0,Y 340.705,Z 161.04,A -85,B 0,C 180,E1 -14196.926,E2 -14196.926} C_VEL
LIN {X 0,Y 340.713,Z 161.044,A -85,B 0,C 180,E1 -14200.729,E2 -14200.729} C_VEL
LIN {X 0,Y 340.797,Z 161.033,A -85,B 0,C 180,E1 -14204.45,E2 -14204.45} C_VEL
LIN {X 0,Y 340.853,Z 161.027,A -85,B 0,C 180,E1 -14208.101,E2 -14208.101} C_VEL
LIN {X 0,Y 340.984,Z 161.013,A -85,B 0,C 180,E1 -14211.705,E2 -14211.705} C_VEL
LIN {X 0,Y 341.019,Z 161.01,A -85,B 0,C 180,E1 -14214.086,E2 -14214.086} C_VEL
LIN {X 0,Y 341.123,Z 161.08,A -85,B 0,C 180,E1 -14218.451,E2 -14218.451} C_VEL
LIN {X 0,Y 343.201,Z 169.105,A -85,B 0,C 180,E1 -14221.174,E2 -14221.174} C_VEL
LIN {X 0,Y 344.072,Z 172.983,A -85,B 0,C 180,E1 -14222.407,E2 -14222.407} C_VEL
LIN {X 0,Y 351.574,Z 189.277,A -85,B 0,C 180,E1 -14223.743,E2 -14223.743} C_VEL
LIN {X 0,Y 353.178,Z 195.142,A -85,B 0,C 180,E1 -14224.083,E2 -14224.083} C_VEL
LIN {X 0,Y 354.579,Z 202.428,A -85,B 0,C 180,E1 -14224.441,E2 -14224.441} C_VEL
LIN {X 0,Y 351.4,Z 281.614,A -85,B 0,C 180,E1 -14226.496,E2 -14226.496} C_VEL
LIN {X 0,Y 350.59,Z 294.631,A -85,B 0,C 180,E1 -14227.053,E2 -14227.053} C_VEL
LIN {X 0,Y 349.583,Z 306.878,A -85,B 0,C 180,E1 -14227.8,E2 -14227.8} C_VEL
LIN {X 0,Y 348.431,Z 318.51,A -85,B 0,C 180,E1 -14228.749,E2 -14228.749} C_VEL
LIN {X 0,Y 347.011,Z 329.8,A -85,B 0,C 180,E1 -14229.913,E2 -14229.913} C_VEL
LIN {X 0,Y 345.553,Z 340.397,A -85,B 0,C 180,E1 -14231.289,E2 -14231.289} C_VEL
LIN {X 0,Y 344.223,Z 348.968,A -85,B 0,C 180,E1 -14232.661,E2 -14232.661} C_VEL
LIN {X 0,Y 342.837,Z 358.117,A -85,B 0,C 180,E1 -14234.48,E2 -14234.48} C_VEL
LIN {X 0,Y 341.762,Z 364.776,A -85,B 0,C 180,E1 -14236.118,E2 -14236.118} C_VEL
LIN {X 0,Y 340.772,Z 370.913,A -85,B 0,C 180,E1 -14238.021,E2 -14238.021} C_VEL
LIN {X 0,Y 340.072,Z 375.644,A -85,B 0,C 180,E1 -14239.938,E2 -14239.938} C_VEL
LIN {X 0,Y 339.543,Z 379.146,A -85,B 0,C 180,E1 -14241.875,E2 -14241.875} C_VEL
LIN {X 0,Y 339.283,Z 380.853,A -85,B 0,C 180,E1 -14243.177,E2 -14243.177} C_VEL
LIN {X 0,Y 339.089,Z 382.007,A -85,B 0,C 180,E1 -14244.49,E2 -14244.49} C_VEL
LIN {X 0,Y 338.912,Z 382.684,A -85,B 0,C 180,E1 -14245.816,E2 -14245.816} C_VEL
LIN {X 0,Y 338.835,Z 382.842,A -85,B 0,C 180,E1 -14247.15,E2 -14247.15} C_VEL
LIN {X 0,Y 338.829,Z 381.894,A -85,B 0,C 180,E1 -14249.404,E2 -14249.404} C_VEL
LIN {X 0,Y 339.005,Z 379.256,A -85,B 0,C 180,E1 -14251.789,E2 -14251.789} C_VEL
LIN {X 0,Y 339.228,Z 376.645,A -85,B 0,C 180,E1 -14253.3,E2 -14253.3} C_VEL
LIN {X 0,Y 339.51,Z 371.646,A -85,B 0,C 180,E1 -14255.424,E2 -14255.424} C_VEL
LIN {X 0,Y 339.996,Z 366.122,A -85,B 0,C 180,E1 -14257.202,E2 -14257.202} C_VEL
LIN {X 0,Y 340.595,Z 359.102,A -85,B 0,C 180,E1 -14259.002,E2 -14259.002} C_VEL
LIN {X 0,Y 341.356,Z 350.811,A -85,B 0,C 180,E1 -14260.712,E2 -14260.712} C_VEL
LIN {X 0,Y 342.198,Z 341.067,A -85,B 0,C 180,E1 -14262.322,E2 -14262.322} C_VEL
LIN {X 0,Y 343.13,Z 330.507,A -85,B 0,C 180,E1 -14263.731,E2 -14263.731} C_VEL
LIN {X 0,Y 344.152,Z 318.604,A -85,B 0,C 180,E1 -14264.984,E2 -14264.984} C_VEL
LIN {X 0,Y 345.027,Z 306.564,A -85,B 0,C 180,E1 -14265.974,E2 -14265.974} C_VEL
LIN {X 0,Y 345.744,Z 293.492,A -85,B 0,C 180,E1 -14266.777,E2 -14266.777} C_VEL
LIN {X 0,Y 346.244,Z 280.686,A -85,B 0,C 180,E1 -14267.322,E2 -14267.322} C_VEL
LIN {X 0,Y 346.842,Z 257.557,A -85,B 0,C 180,E1 -14267.914,E2 -14267.914} C_VEL
LIN {X 0,Y 348.348,Z 198.894,A -85,B 0,C 180,E1 -14269.336,E2 -14269.336} C_VEL
LIN {X 0,Y 344.274,Z 176.547,A -85,B 0,C 180,E1 -14270.123,E2 -14270.123} C_VEL
LIN {X 0,Y 342.748,Z 171.572,A -85,B 0,C 180,E1 -14270.34,E2 -14270.34} C_VEL
LIN {X 0,Y 340.777,Z 161.038,A -85,B 0,C 180,E1 -14273.462,E2 -14273.462} C_VEL
LIN {X 0,Y 340.698,Z 161.045,A -85,B 0,C 180,E1 -14276.153,E2 -14276.153} C_VEL
LIN {X 0,Y 340.724,Z 161.042,A -85,B 0,C 180,E1 -14280.035,E2 -14280.035} C_VEL
LIN {X 0,Y 340.714,Z 161.042,A -85,B 0,C 180,E1 -14283.011,E2 -14283.011} C_VEL
LIN {X 0,Y 340.705,Z 161.043,A -85,B 0,C 180,E1 -14286.924,E2 -14286.924} C_VEL
LIN {X 0,Y 340.704,Z 161.044,A -85,B 0,C 180,E1 -14290.727,E2 -14290.727} C_VEL
LIN {X 0,Y 340.794,Z 161.034,A -85,B 0,C 180,E1 -14294.448,E2 -14294.448} C_VEL
LIN {X 0,Y 340.85,Z 161.03,A -85,B 0,C 180,E1 -14298.1,E2 -14298.1} C_VEL
LIN {X 0,Y 340.985,Z 161.01,A -85,B 0,C 180,E1 -14301.704,E2 -14301.704} C_VEL
LIN {X 0,Y 341.016,Z 161.008,A -85,B 0,C 180,E1 -14304.084,E2 -14304.084} C_VEL
LIN {X 0,Y 341.128,Z 160.993,A -85,B 0,C 180,E1 -14307.637,E2 -14307.637} C_VEL
LIN {X 0,Y 341.091,Z 160.995,A -85,B 0,C 180,E1 -14311.18,E2 -14311.18} C_VEL
LIN {X 0,Y 341.128,Z 160.99,A -85,B 0,C 180,E1 -14312.36,E2 -14312.36} C_VEL
LIN {X 0,Y 341.002,Z 161.006,A -85,B 0,C 180,E1 -14317.102,E2 -14317.102} C_VEL
LIN {X 0,Y 340.846,Z 161.024,A -85,B 0,C 180,E1 -14320.693,E2 -14320.693} C_VEL
LIN {X 0,Y 340.82,Z 161.028,A -85,B 0,C 180,E1 -14324.326,E2 -14324.326} C_VEL
LIN {X 0,Y 340.756,Z 161.036,A -85,B 0,C 180,E1 -14328.423,E2 -14328.423} C_VEL
LIN {X 0,Y 340.712,Z 161.042,A -85,B 0,C 180,E1 -14331.942,E2 -14331.942} C_VEL
LIN {X 0,Y 340.67,Z 161.049,A -85,B 0,C 180,E1 -14335.671,E2 -14335.671} C_VEL
LIN {X 0,Y 340.704,Z 161.045,A -85,B 0,C 180,E1 -14337.085,E2 -14337.085} C_VEL
LIN {X 0,Y 339.997,Z 161.132,A -85,B 0,C 180,E1 -14338.072,E2 -14338.072} C_VEL
LIN {X 0,Y 337.115,Z 161.491,A -85,B 0,C 180,E1 -14339.678,E2 -14339.678} C_VEL
LIN {X 0,Y 334.709,Z 161.793,A -85,B 0,C 180,E1 -14340.978,E2 -14340.978} C_VEL
LIN {X 0,Y 333.701,Z 161.915,A -85,B 0,C 180,E1 -14341.984,E2 -14341.984} C_VEL
LIN {X 0,Y 333.63,Z 161.924,A -85,B 0,C 180,E1 -14342.325,E2 -14342.325} C_VEL
LIN {X 0,Y 333.672,Z 161.918,A -85,B 0,C 180,E1 -14346.138,E2 -14346.138} C_VEL
LIN {X 0,Y 333.618,Z 161.929,A -85,B 0,C 180,E1 -14349.195,E2 -14349.195} C_VEL
LIN {X 0,Y 333.625,Z 161.926,A -85,B 0,C 180,E1 -14352.498,E2 -14352.498} C_VEL
LIN {X 0,Y 333.59,Z 161.928,A -85,B 0,C 180,E1 -14355.953,E2 -14355.953} C_VEL
LIN {X 0,Y 333.598,Z 161.929,A -85,B 0,C 180,E1 -14359.323,E2 -14359.323} C_VEL
LIN {X 0,Y 333.658,Z 161.922,A -85,B 0,C 180,E1 -14363.167,E2 -14363.167} C_VEL
LIN {X 0,Y 333.669,Z 161.919,A -85,B 0,C 180,E1 -14365.34,E2 -14365.34} C_VEL
LIN {X 0,Y 333.624,Z 161.926,A -85,B 0,C 180,E1 -14368.221,E2 -14368.221} C_VEL
LIN {X 0,Y 333.646,Z 161.923,A -85,B 0,C 180,E1 -14371.021,E2 -14371.021} C_VEL
LIN {X 0,Y 333.655,Z 161.921,A -85,B 0,C 180,E1 -14375.084,E2 -14375.084} C_VEL
LIN {X 0,Y 333.646,Z 161.922,A -85,B 0,C 180,E1 -14379.016,E2 -14379.016} C_VEL
LIN {X 0,Y 333.706,Z 161.914,A -85,B 0,C 180,E1 -14381.584,E2 -14381.584} C_VEL
LIN {X 0,Y 333.767,Z 161.907,A -85,B 0,C 180,E1 -14385.6,E2 -14385.6} C_VEL
LIN {X 0,Y 333.806,Z 161.901,A -85,B 0,C 180,E1 -14389.077,E2 -14389.077} C_VEL
LIN {X 0,Y 333.949,Z 161.884,A -85,B 0,C 180,E1 -14392.746,E2 -14392.746} C_VEL
LIN {X 0,Y 333.77,Z 161.906,A -85,B 0,C 180,E1 -14395.168,E2 -14395.168} C_VEL
LIN {X 0,Y 334.057,Z 161.872,A -85,B 0,C 180,E1 -14397.588,E2 -14397.588} C_VEL
LIN {X 0,Y 334.05,Z 161.872,A -85,B 0,C 180,E1 -14401.205,E2 -14401.205} C_VEL
LIN {X 0,Y 334.057,Z 161.872,A -85,B 0,C 180,E1 -14402.411,E2 -14402.411} C_VEL
LIN {X 0,Y 333.98,Z 161.883,A -85,B 0,C 180,E1 -14406.039,E2 -14406.039} C_VEL
LIN {X 0,Y 333.905,Z 161.89,A -85,B 0,C 180,E1 -14408.472,E2 -14408.472} C_VEL
LIN {X 0,Y 333.779,Z 161.907,A -85,B 0,C 180,E1 -14412.155,E2 -14412.155} C_VEL
LIN {X 0,Y 333.743,Z 161.909,A -85,B 0,C 180,E1 -14414.637,E2 -14414.637} C_VEL
LIN {X 0,Y 333.685,Z 161.916,A -85,B 0,C 180,E1 -14418.602,E2 -14418.602} C_VEL
LIN {X 0,Y 333.641,Z 161.922,A -85,B 0,C 180,E1 -14422.282,E2 -14422.282} C_VEL
LIN {X 0,Y 333.65,Z 161.923,A -85,B 0,C 180,E1 -14425.078,E2 -14425.078} C_VEL
LIN {X 0,Y 333.641,Z 161.924,A -85,B 0,C 180,E1 -14428.979,E2 -14428.979} C_VEL
LIN {X 0,Y 333.637,Z 161.923,A -85,B 0,C 180,E1 -14432.587,E2 -14432.587} C_VEL
LIN {X 0,Y 333.666,Z 161.919,A -85,B 0,C 180,E1 -14436.14,E2 -14436.14} C_VEL
LIN {X 0,Y 333.613,Z 161.931,A -85,B 0,C 180,E1 -14439.197,E2 -14439.197} C_VEL
LIN {X 0,Y 333.62,Z 161.926,A -85,B 0,C 180,E1 -14442.499,E2 -14442.499} C_VEL
LIN {X 0,Y 333.588,Z 161.929,A -85,B 0,C 180,E1 -14445.955,E2 -14445.955} C_VEL
LIN {X 0,Y 333.596,Z 161.93,A -85,B 0,C 180,E1 -14449.326,E2 -14449.326} C_VEL
LIN {X 0,Y 333.657,Z 161.923,A -85,B 0,C 180,E1 -14453.17,E2 -14453.17} C_VEL
LIN {X 0,Y 333.668,Z 161.92,A -85,B 0,C 180,E1 -14455.342,E2 -14455.342} C_VEL
LIN {X 0,Y 333.625,Z 161.925,A -85,B 0,C 180,E1 -14458.223,E2 -14458.223} C_VEL
LIN {X 0,Y 333.689,Z 161.967,A -85,B 0,C 180,E1 -14459.983,E2 -14459.983} C_VEL
LIN {X 0,Y 336.297,Z 175.173,A -85,B 0,C 180,E1 -14463.637,E2 -14463.637} C_VEL
LIN {X 0,Y 337.156,Z 180.384,A -85,B 0,C 180,E1 -14465.033,E2 -14465.033} C_VEL
LIN {X 0,Y 336.551,Z 187.737,A -85,B 0,C 180,E1 -14466.879,E2 -14466.879} C_VEL
LIN {X 0,Y 336.338,Z 189.862,A -85,B 0,C 180,E1 -14467.349,E2 -14467.349} C_VEL
LIN {X 0,Y 341.137,Z 225.78,A -85,B 0,C 180,E1 -14468.549,E2 -14468.549} C_VEL
LIN {X 0,Y 339.328,Z 298.206,A -85,B 0,C 180,E1 -14470.373,E2 -14470.373} C_VEL
LIN {X 0,Y 338.631,Z 312.056,A -85,B 0,C 180,E1 -14470.961,E2 -14470.961} C_VEL
LIN {X 0,Y 337.785,Z 324.632,A -85,B 0,C 180,E1 -14471.737,E2 -14471.737} C_VEL
LIN {X 0,Y 336.879,Z 336.334,A -85,B 0,C 180,E1 -14472.707,E2 -14472.707} C_VEL
LIN {X 0,Y 335.816,Z 347.714,A -85,B 0,C 180,E1 -14473.902,E2 -14473.902} C_VEL
LIN {X 0,Y 334.968,Z 357.791,A -85,B 0,C 180,E1 -14475.227,E2 -14475.227} C_VEL
LIN {X 0,Y 333.996,Z 368.146,A -85,B 0,C 180,E1 -14476.927,E2 -14476.927} C_VEL
LIN {X 0,Y 333.097,Z 377.021,A -85,B 0,C 180,E1 -14478.747,E2 -14478.747} C_VEL
LIN {X 0,Y 332.578,Z 384.088,A -85,B 0,C 180,E1 -14480.575,E2 -14480.575} C_VEL
LIN {X 0,Y 332.191,Z 390.551,A -85,B 0,C 180,E1 -14482.708,E2 -14482.708} C_VEL
LIN {X 0,Y 332.026,Z 393.987,A -85,B 0,C 180,E1 -14484.182,E2 -14484.182} C_VEL
LIN {X 0,Y 332.004,Z 397.783,A -85,B 0,C 180,E1 -14486.36,E2 -14486.36} C_VEL
LIN {X 0,Y 331.927,Z 399.231,A -85,B 0,C 180,E1 -14487.574,E2 -14487.574} C_VEL
LIN {X 0,Y 331.932,Z 400.241,A -85,B 0,C 180,E1 -14488.788,E2 -14488.788} C_VEL
LIN {X 0,Y 331.974,Z 400.842,A -85,B 0,C 180,E1 -14490.001,E2 -14490.001} C_VEL
LIN {X 0,Y 331.912,Z 401.022,A -85,B 0,C 180,E1 -14491.214,E2 -14491.214} C_VEL
LIN {X 0,Y 331.913,Z 400.746,A -85,B 0,C 180,E1 -14492.428,E2 -14492.428} C_VEL
LIN {X 0,Y 331.967,Z 400.062,A -85,B 0,C 180,E1 -14493.642,E2 -14493.642} C_VEL
LIN {X 0,Y 332.005,Z 397.848,A -85,B 0,C 180,E1 -14495.782,E2 -14495.782} C_VEL
LIN {X 0,Y 332.374,Z 394.319,A -85,B 0,C 180,E1 -14497.901,E2 -14497.901} C_VEL
LIN {X 0,Y 332.874,Z 390.108,A -85,B 0,C 180,E1 -14499.725,E2 -14499.725} C_VEL
LIN {X 0,Y 333.752,Z 383.677,A -85,B 0,C 180,E1 -14501.849,E2 -14501.849} C_VEL
LIN {X 0,Y 334.931,Z 376.726,A -85,B 0,C 180,E1 -14503.655,E2 -14503.655} C_VEL
LIN {X 0,Y 336.343,Z 368.106,A -85,B 0,C 180,E1 -14505.452,E2 -14505.452} C_VEL
LIN {X 0,Y 337.548,Z 359.299,A -85,B 0,C 180,E1 -14506.948,E2 -14506.948} C_VEL
LIN {X 0,Y 339.271,Z 348.504,A -85,B 0,C 180,E1 -14508.416,E2 -14508.416} C_VEL
LIN {X 0,Y 340.826,Z 337.837,A -85,B 0,C 180,E1 -14509.579,E2 -14509.579} C_VEL
LIN {X 0,Y 342.234,Z 326.076,A -85,B 0,C 180,E1 -14510.591,E2 -14510.591} C_VEL
LIN {X 0,Y 343.452,Z 314.249,A -85,B 0,C 180,E1 -14511.377,E2 -14511.377} C_VEL
LIN {X 0,Y 344.692,Z 300.888,A -85,B 0,C 180,E1 -14512.004,E2 -14512.004} C_VEL
LIN {X 0,Y 345.457,Z 284.159,A -85,B 0,C 180,E1 -14512.503,E2 -14512.503} C_VEL
LIN {X 0,Y 347.521,Z 226.331,A -85,B 0,C 180,E1 -14514.04,E2 -14514.04} C_VEL
LIN {X 0,Y 344.774,Z 208.901,A -85,B 0,C 180,E1 -14514.863,E2 -14514.863} C_VEL
LIN {X 0,Y 340.696,Z 190.473,A -85,B 0,C 180,E1 -14515.914,E2 -14515.914} C_VEL
LIN {X 0,Y 339.497,Z 187.154,A -85,B 0,C 180,E1 -14516.173,E2 -14516.173} C_VEL
LIN {X 0,Y 337.728,Z 177.52,A -85,B 0,C 180,E1 -14519.073,E2 -14519.073} C_VEL
LIN {X 0,Y 335.863,Z 169.941,A -85,B 0,C 180,E1 -14521.543,E2 -14521.543} C_VEL
LIN {X 0,Y 333.678,Z 161.922,A -85,B 0,C 180,E1 -14524.385,E2 -14524.385} C_VEL
LIN {X 0,Y 333.645,Z 161.923,A -85,B 0,C 180,E1 -14527.653,E2 -14527.653} C_VEL
LIN {X 0,Y 333.606,Z 161.93,A -85,B 0,C 180,E1 -14530.775,E2 -14530.775} C_VEL
LIN {X 0,Y 333.593,Z 161.928,A -85,B 0,C 180,E1 -14534.25,E2 -14534.25} C_VEL
LIN {X 0,Y 333.64,Z 161.92,A -85,B 0,C 180,E1 -14537.618,E2 -14537.618} C_VEL
LIN {X 0,Y 333.619,Z 161.92,A -85,B 0,C 180,E1 -14541.211,E2 -14541.211} C_VEL
LIN {X 0,Y 333.676,Z 161.915,A -85,B 0,C 180,E1 -14543.861,E2 -14543.861} C_VEL
LIN {X 0,Y 333.647,Z 161.924,A -85,B 0,C 180,E1 -14547.414,E2 -14547.414} C_VEL
LIN {X 0,Y 333.655,Z 161.92,A -85,B 0,C 180,E1 -14551.023,E2 -14551.023} C_VEL
LIN {X 0,Y 333.668,Z 161.92,A -85,B 0,C 180,E1 -14555.086,E2 -14555.086} C_VEL
LIN {X 0,Y 333.658,Z 161.917,A -85,B 0,C 180,E1 -14559.018,E2 -14559.018} C_VEL
LIN {X 0,Y 333.717,Z 161.913,A -85,B 0,C 180,E1 -14561.585,E2 -14561.585} C_VEL
LIN {X 0,Y 333.778,Z 161.909,A -85,B 0,C 180,E1 -14565.601,E2 -14565.601} C_VEL
LIN {X 0,Y 333.821,Z 161.906,A -85,B 0,C 180,E1 -14569.078,E2 -14569.078} C_VEL
LIN {X 0,Y 333.961,Z 161.889,A -85,B 0,C 180,E1 -14572.746,E2 -14572.746} C_VEL
LIN {X 0,Y 333.784,Z 161.908,A -85,B 0,C 180,E1 -14575.169,E2 -14575.169} C_VEL
LIN {X 0,Y 334.094,Z 161.903,A -85,B 0,C 180,E1 -14577.589,E2 -14577.589} C_VEL
LIN {X 0,Y 336.333,Z 170.372,A -85,B 0,C 180,E1 -14580.599,E2 -14580.599} C_VEL
LIN {X 0,Y 337.118,Z 173.496,A -85,B 0,C 180,E1 -14581.6,E2 -14581.6} C_VEL
LIN {X 0,Y 345.558,Z 191.52,A -85,B 0,C 180,E1 -14583.177,E2 -14583.177} C_VEL
LIN {X 0,Y 346.667,Z 194.785,A -85,B 0,C 180,E1 -14583.403,E2 -14583.403} C_VEL
LIN {X 0,Y 348.454,Z 203.381,A -85,B 0,C 180,E1 -14583.856,E2 -14583.856} C_VEL
LIN {X 0,Y 345.137,Z 282.191,A -85,B 0,C 180,E1 -14585.954,E2 -14585.954} C_VEL
LIN {X 0,Y 344.287,Z 295.003,A -85,B 0,C 180,E1 -14586.52,E2 -14586.52} C_VEL
LIN {X 0,Y 343.244,Z 307.11,A -85,B 0,C 180,E1 -14587.279,E2 -14587.279} C_VEL
LIN {X 0,Y 341.951,Z 319.002,A -85,B 0,C 180,E1 -14588.272,E2 -14588.272} C_VEL
LIN {X 0,Y 340.402,Z 330.691,A -85,B 0,C 180,E1 -14589.507,E2 -14589.507} C_VEL
LIN {X 0,Y 338.886,Z 341.135,A -85,B 0,C 180,E1 -14590.909,E2 -14590.909} C_VEL
LIN {X 0,Y 337.256,Z 351.11,A -85,B 0,C 180,E1 -14592.578,E2 -14592.578} C_VEL
LIN {X 0,Y 335.968,Z 359.03,A -85,B 0,C 180,E1 -14594.229,E2 -14594.229} C_VEL
LIN {X 0,Y 334.696,Z 366.38,A -85,B 0,C 180,E1 -14596.155,E2 -14596.155} C_VEL
LIN {X 0,Y 333.829,Z 371.334,A -85,B 0,C 180,E1 -14597.774,E2 -14597.774} C_VEL
LIN {X 0,Y 333.072,Z 376.014,A -85,B 0,C 180,E1 -14599.732,E2 -14599.732} C_VEL
LIN {X 0,Y 332.532,Z 379.275,A -85,B 0,C 180,E1 -14601.574,E2 -14601.574} C_VEL
LIN {X 0,Y 332.106,Z 381.767,A -85,B 0,C 180,E1 -14603.709,E2 -14603.709} C_VEL
LIN {X 0,Y 331.911,Z 382.67,A -85,B 0,C 180,E1 -14605.055,E2 -14605.055} C_VEL
LIN {X 0,Y 331.737,Z 383.024,A -85,B 0,C 180,E1 -14607.152,E2 -14607.152} C_VEL
LIN {X 0,Y 331.745,Z 381.811,A -85,B 0,C 180,E1 -14609.704,E2 -14609.704} C_VEL
LIN {X 0,Y 331.937,Z 379.128,A -85,B 0,C 180,E1 -14611.96,E2 -14611.96} C_VEL
LIN {X 0,Y 332.208,Z 375.589,A -85,B 0,C 180,E1 -14613.902,E2 -14613.902} C_VEL
LIN {X 0,Y 332.517,Z 370.604,A -85,B 0,C 180,E1 -14615.911,E2 -14615.911} C_VEL
LIN {X 0,Y 333.056,Z 364.761,A -85,B 0,C 180,E1 -14617.731,E2 -14617.731} C_VEL
LIN {X 0,Y 333.705,Z 357.285,A -85,B 0,C 180,E1 -14619.575,E2 -14619.575} C_VEL
LIN {X 0,Y 334.651,Z 347.807,A -85,B 0,C 180,E1 -14621.44,E2 -14621.44} C_VEL
LIN {X 0,Y 335.498,Z 338.281,A -85,B 0,C 180,E1 -14622.944,E2 -14622.944} C_VEL
LIN {X 0,Y 336.522,Z 326.781,A -85,B 0,C 180,E1 -14624.397,E2 -14624.397} C_VEL
LIN {X 0,Y 337.472,Z 315.789,A -85,B 0,C 180,E1 -14625.503,E2 -14625.503} C_VEL
LIN {X 0,Y 338.288,Z 303.93,A -85,B 0,C 180,E1 -14626.431,E2 -14626.431} C_VEL
LIN {X 0,Y 338.993,Z 290.391,A -85,B 0,C 180,E1 -14627.219,E2 -14627.219} C_VEL
LIN {X 0,Y 339.525,Z 277.212,A -85,B 0,C 180,E1 -14627.725,E2 -14627.725} C_VEL
LIN {X 0,Y 341.548,Z 199.738,A -85,B 0,C 180,E1 -14629.652,E2 -14629.652} C_VEL
LIN {X 0,Y 337.686,Z 178.534,A -85,B 0,C 180,E1 -14630.416,E2 -14630.416} C_VEL
LIN {X 0,Y 335.585,Z 171.716,A -85,B 0,C 180,E1 -14630.729,E2 -14630.729} C_VEL
LIN {X 0,Y 333.717,Z 161.917,A -85,B 0,C 180,E1 -14633.656,E2 -14633.656} C_VEL
LIN {X 0,Y 333.649,Z 161.921,A -85,B 0,C 180,E1 -14637.413,E2 -14637.413} C_VEL
LIN {X 0,Y 333.633,Z 161.924,A -85,B 0,C 180,E1 -14641.02,E2 -14641.02} C_VEL
LIN {X 0,Y 333.661,Z 161.921,A -85,B 0,C 180,E1 -14644.922,E2 -14644.922} C_VEL
LIN {X 0,Y 333.654,Z 161.921,A -85,B 0,C 180,E1 -14649.016,E2 -14649.016} C_VEL
LIN {X 0,Y 333.715,Z 161.914,A -85,B 0,C 180,E1 -14651.584,E2 -14651.584} C_VEL
LIN {X 0,Y 333.779,Z 161.906,A -85,B 0,C 180,E1 -14655.599,E2 -14655.599} C_VEL
LIN {X 0,Y 333.819,Z 161.9,A -85,B 0,C 180,E1 -14659.077,E2 -14659.077} C_VEL
LIN {X 0,Y 333.96,Z 161.883,A -85,B 0,C 180,E1 -14662.745,E2 -14662.745} C_VEL
LIN {X 0,Y 333.779,Z 161.905,A -85,B 0,C 180,E1 -14665.168,E2 -14665.168} C_VEL
LIN {X 0,Y 334.068,Z 161.872,A -85,B 0,C 180,E1 -14667.588,E2 -14667.588} C_VEL
LIN {X 0,Y 334.062,Z 161.871,A -85,B 0,C 180,E1 -14671.204,E2 -14671.204} C_VEL
LIN {X 0,Y 334.068,Z 161.869,A -85,B 0,C 180,E1 -14672.41,E2 -14672.41} C_VEL
LIN {X 0,Y 333.988,Z 161.881,A -85,B 0,C 180,E1 -14676.038,E2 -14676.038} C_VEL
LIN {X 0,Y 333.916,Z 161.888,A -85,B 0,C 180,E1 -14678.471,E2 -14678.471} C_VEL
LIN {X 0,Y 333.789,Z 161.905,A -85,B 0,C 180,E1 -14682.154,E2 -14682.154} C_VEL
LIN {X 0,Y 333.753,Z 161.908,A -85,B 0,C 180,E1 -14684.636,E2 -14684.636} C_VEL
LIN {X 0,Y 333.694,Z 161.916,A -85,B 0,C 180,E1 -14688.601,E2 -14688.601} C_VEL
LIN {X 0,Y 333.65,Z 161.921,A -85,B 0,C 180,E1 -14692.28,E2 -14692.28} C_VEL
LIN {X 0,Y 333.658,Z 161.924,A -85,B 0,C 180,E1 -14695.077,E2 -14695.077} C_VEL
LIN {X 0,Y 333.649,Z 161.925,A -85,B 0,C 180,E1 -14698.977,E2 -14698.977} C_VEL
LIN {X 0,Y 333.63,Z 161.924,A -85,B 0,C 180,E1 -14702.325,E2 -14702.325} C_VEL
LIN {X 0,Y 333,Z 162.006,A -85,B 0,C 180,E1 -14703.333,E2 -14703.333} C_VEL
LIN {X 0,Y 330.178,Z 162.36,A -85,B 0,C 180,E1 -14704.973,E2 -14704.973} C_VEL
LIN {X 0,Y 327.751,Z 162.661,A -85,B 0,C 180,E1 -14706.301,E2 -14706.301} C_VEL
LIN {X 0,Y 326.685,Z 162.792,A -85,B 0,C 180,E1 -14707.328,E2 -14707.328} C_VEL
LIN {X 0,Y 326.587,Z 162.801,A -85,B 0,C 180,E1 -14707.677,E2 -14707.677} C_VEL
LIN {X 0,Y 326.542,Z 162.811,A -85,B 0,C 180,E1 -14711.123,E2 -14711.123} C_VEL
LIN {X 0,Y 326.556,Z 162.805,A -85,B 0,C 180,E1 -14713.525,E2 -14713.525} C_VEL
LIN {X 0,Y 326.569,Z 162.807,A -85,B 0,C 180,E1 -14717.028,E2 -14717.028} C_VEL
LIN {X 0,Y 326.578,Z 162.803,A -85,B 0,C 180,E1 -14721.384,E2 -14721.384} C_VEL
LIN {X 0,Y 326.615,Z 162.801,A -85,B 0,C 180,E1 -14724.85,E2 -14724.85} C_VEL
LIN {X 0,Y 326.603,Z 162.799,A -85,B 0,C 180,E1 -14727.454,E2 -14727.454} C_VEL
LIN {X 0,Y 326.61,Z 162.802,A -85,B 0,C 180,E1 -14730.335,E2 -14730.335} C_VEL
LIN {X 0,Y 326.593,Z 162.805,A -85,B 0,C 180,E1 -14734.508,E2 -14734.508} C_VEL
LIN {X 0,Y 326.602,Z 162.803,A -85,B 0,C 180,E1 -14738.542,E2 -14738.542} C_VEL
LIN {X 0,Y 326.641,Z 162.794,A -85,B 0,C 180,E1 -14741.205,E2 -14741.205} C_VEL
LIN {X 0,Y 326.719,Z 162.785,A -85,B 0,C 180,E1 -14745.459,E2 -14745.459} C_VEL
LIN {X 0,Y 326.748,Z 162.781,A -85,B 0,C 180,E1 -14748.838,E2 -14748.838} C_VEL
LIN {X 0,Y 326.906,Z 162.763,A -85,B 0,C 180,E1 -14752.588,E2 -14752.588} C_VEL
LIN {X 0,Y 326.739,Z 162.782,A -85,B 0,C 180,E1 -14755.064,E2 -14755.064} C_VEL
LIN {X 0,Y 327.001,Z 162.751,A -85,B 0,C 180,E1 -14757.536,E2 -14757.536} C_VEL
LIN {X 0,Y 327.021,Z 162.747,A -85,B 0,C 180,E1 -14761.231,E2 -14761.231} C_VEL
LIN {X 0,Y 326.742,Z 162.786,A -85,B 0,C 180,E1 -14763.699,E2 -14763.699} C_VEL
LIN {X 0,Y 326.934,Z 162.76,A -85,B 0,C 180,E1 -14766.17,E2 -14766.17} C_VEL
LIN {X 0,Y 326.774,Z 162.782,A -85,B 0,C 180,E1 -14769.907,E2 -14769.907} C_VEL
LIN {X 0,Y 326.735,Z 162.788,A -85,B 0,C 180,E1 -14773.686,E2 -14773.686} C_VEL
LIN {X 0,Y 326.619,Z 162.802,A -85,B 0,C 180,E1 -14777.532,E2 -14777.532} C_VEL
LIN {X 0,Y 326.594,Z 162.805,A -85,B 0,C 180,E1 -14781.458,E2 -14781.458} C_VEL
LIN {X 0,Y 326.592,Z 162.805,A -85,B 0,C 180,E1 -14785.492,E2 -14785.492} C_VEL
LIN {X 0,Y 326.606,Z 162.801,A -85,B 0,C 180,E1 -14789.664,E2 -14789.664} C_VEL
LIN {X 0,Y 326.61,Z 162.801,A -85,B 0,C 180,E1 -14792.946,E2 -14792.946} C_VEL
LIN {X 0,Y 326.604,Z 162.801,A -85,B 0,C 180,E1 -14795.521,E2 -14795.521} C_VEL
LIN {X 0,Y 326.581,Z 162.806,A -85,B 0,C 180,E1 -14799.223,E2 -14799.223} C_VEL
LIN {X 0,Y 326.566,Z 162.808,A -85,B 0,C 180,E1 -14802.972,E2 -14802.972} C_VEL
LIN {X 0,Y 326.566,Z 162.809,A -85,B 0,C 180,E1 -14807.03,E2 -14807.03} C_VEL
LIN {X 0,Y 326.577,Z 162.803,A -85,B 0,C 180,E1 -14811.386,E2 -14811.386} C_VEL
LIN {X 0,Y 326.614,Z 162.803,A -85,B 0,C 180,E1 -14814.853,E2 -14814.853} C_VEL
LIN {X 0,Y 326.604,Z 162.799,A -85,B 0,C 180,E1 -14817.457,E2 -14817.457} C_VEL
LIN {X 0,Y 326.632,Z 162.914,A -85,B 0,C 180,E1 -14819.73,E2 -14819.73} C_VEL
LIN {X 0,Y 329.172,Z 175.753,A -85,B 0,C 180,E1 -14823.363,E2 -14823.363} C_VEL
LIN {X 0,Y 330.162,Z 182.283,A -85,B 0,C 180,E1 -14825.141,E2 -14825.141} C_VEL
LIN {X 0,Y 329.436,Z 189.401,A -85,B 0,C 180,E1 -14826.961,E2 -14826.961} C_VEL
LIN {X 0,Y 334.297,Z 226.364,A -85,B 0,C 180,E1 -14828.227,E2 -14828.227} C_VEL
LIN {X 0,Y 332.42,Z 298.668,A -85,B 0,C 180,E1 -14830.109,E2 -14830.109} C_VEL
LIN {X 0,Y 331.696,Z 312.274,A -85,B 0,C 180,E1 -14830.708,E2 -14830.708} C_VEL
LIN {X 0,Y 330.926,Z 323.689,A -85,B 0,C 180,E1 -14831.425,E2 -14831.425} C_VEL
LIN {X 0,Y 329.91,Z 336.342,A -85,B 0,C 180,E1 -14832.489,E2 -14832.489} C_VEL
LIN {X 0,Y 328.822,Z 347.68,A -85,B 0,C 180,E1 -14833.71,E2 -14833.71} C_VEL
LIN {X 0,Y 327.924,Z 357.956,A -85,B 0,C 180,E1 -14835.098,E2 -14835.098} C_VEL
LIN {X 0,Y 327.016,Z 367.221,A -85,B 0,C 180,E1 -14836.643,E2 -14836.643} C_VEL
LIN {X 0,Y 326.1,Z 376.251,A -85,B 0,C 180,E1 -14838.502,E2 -14838.502} C_VEL
LIN {X 0,Y 325.536,Z 383.442,A -85,B 0,C 180,E1 -14840.369,E2 -14840.369} C_VEL
LIN {X 0,Y 325.141,Z 389.995,A -85,B 0,C 180,E1 -14842.549,E2 -14842.549} C_VEL
LIN {X 0,Y 324.925,Z 393.906,A -85,B 0,C 180,E1 -14844.246,E2 -14844.246} C_VEL
LIN {X 0,Y 324.931,Z 397.391,A -85,B 0,C 180,E1 -14846.281,E2 -14846.281} C_VEL
LIN {X 0,Y 324.847,Z 398.91,A -85,B 0,C 180,E1 -14847.521,E2 -14847.521} C_VEL
LIN {X 0,Y 324.84,Z 399.956,A -85,B 0,C 180,E1 -14848.761,E2 -14848.761} C_VEL
LIN {X 0,Y 324.878,Z 400.59,A -85,B 0,C 180,E1 -14850.001,E2 -14850.001} C_VEL
LIN {X 0,Y 324.821,Z 400.812,A -85,B 0,C 180,E1 -14851.241,E2 -14851.241} C_VEL
LIN {X 0,Y 324.833,Z 400.592,A -85,B 0,C 180,E1 -14852.481,E2 -14852.481} C_VEL
LIN {X 0,Y 324.873,Z 399.938,A -85,B 0,C 180,E1 -14853.722,E2 -14853.722} C_VEL
LIN {X 0,Y 324.909,Z 398.015,A -85,B 0,C 180,E1 -14855.725,E2 -14855.725} C_VEL
LIN {X 0,Y 325.33,Z 394.337,A -85,B 0,C 180,E1 -14858.073,E2 -14858.073} C_VEL
LIN {X 0,Y 325.853,Z 390.216,A -85,B 0,C 180,E1 -14859.937,E2 -14859.937} C_VEL
LIN {X 0,Y 326.79,Z 383.907,A -85,B 0,C 180,E1 -14862.105,E2 -14862.105} C_VEL
LIN {X 0,Y 328.052,Z 377.038,A -85,B 0,C 180,E1 -14863.947,E2 -14863.947} C_VEL
LIN {X 0,Y 329.52,Z 368.554,A -85,B 0,C 180,E1 -14865.78,E2 -14865.78} C_VEL
LIN {X 0,Y 330.797,Z 359.881,A -85,B 0,C 180,E1 -14867.305,E2 -14867.305} C_VEL
LIN {X 0,Y 332.603,Z 349.286,A -85,B 0,C 180,E1 -14868.799,E2 -14868.799} C_VEL
LIN {X 0,Y 334.211,Z 338.908,A -85,B 0,C 180,E1 -14869.982,E2 -14869.982} C_VEL
LIN {X 0,Y 335.689,Z 327.666,A -85,B 0,C 180,E1 -14871.011,E2 -14871.011} C_VEL
LIN {X 0,Y 337.068,Z 315.136,A -85,B 0,C 180,E1 -14871.883,E2 -14871.883} C_VEL
LIN {X 0,Y 338.434,Z 301.442,A -85,B 0,C 180,E1 -14872.553,E2 -14872.553} C_VEL
LIN {X 0,Y 339.171,Z 286.554,A -85,B 0,C 180,E1 -14873.025,E2 -14873.025} C_VEL
LIN {X 0,Y 341.467,Z 227.482,A -85,B 0,C 180,E1 -14874.626,E2 -14874.626} C_VEL
LIN {X 0,Y 338.958,Z 210.996,A -85,B 0,C 180,E1 -14875.442,E2 -14875.442} C_VEL
LIN {X 0,Y 335.209,Z 193.804,A -85,B 0,C 180,E1 -14876.452,E2 -14876.452} C_VEL
LIN {X 0,Y 333.338,Z 189.306,A -85,B 0,C 180,E1 -14876.839,E2 -14876.839} C_VEL
LIN {X 0,Y 332.415,Z 186.768,A -85,B 0,C 180,E1 -14877.076,E2 -14877.076} C_VEL
LIN {X 0,Y 330.355,Z 176.452,A -85,B 0,C 180,E1 -14880.349,E2 -14880.349} C_VEL
LIN {X 0,Y 328.054,Z 167.989,A -85,B 0,C 180,E1 -14883.331,E2 -14883.331} C_VEL
LIN {X 0,Y 326.634,Z 162.798,A -85,B 0,C 180,E1 -14885.34,E2 -14885.34} C_VEL
LIN {X 0,Y 326.59,Z 162.805,A -85,B 0,C 180,E1 -14889.223,E2 -14889.223} C_VEL
LIN {X 0,Y 326.575,Z 162.804,A -85,B 0,C 180,E1 -14892.972,E2 -14892.972} C_VEL
LIN {X 0,Y 326.576,Z 162.798,A -85,B 0,C 180,E1 -14897.029,E2 -14897.029} C_VEL
LIN {X 0,Y 326.574,Z 162.799,A -85,B 0,C 180,E1 -14900.782,E2 -14900.782} C_VEL
LIN {X 0,Y 326.614,Z 162.796,A -85,B 0,C 180,E1 -14904.481,E2 -14904.481} C_VEL
LIN {X 0,Y 326.611,Z 162.801,A -85,B 0,C 180,E1 -14907.456,E2 -14907.456} C_VEL
LIN {X 0,Y 326.619,Z 162.8,A -85,B 0,C 180,E1 -14910.337,E2 -14910.337} C_VEL
LIN {X 0,Y 326.604,Z 162.796,A -85,B 0,C 180,E1 -14914.509,E2 -14914.509} C_VEL
LIN {X 0,Y 326.613,Z 162.797,A -85,B 0,C 180,E1 -14918.543,E2 -14918.543} C_VEL
LIN {X 0,Y 326.652,Z 162.794,A -85,B 0,C 180,E1 -14921.206,E2 -14921.206} C_VEL
LIN {X 0,Y 326.729,Z 162.788,A -85,B 0,C 180,E1 -14925.46,E2 -14925.46} C_VEL
LIN {X 0,Y 326.762,Z 162.785,A -85,B 0,C 180,E1 -14928.839,E2 -14928.839} C_VEL
LIN {X 0,Y 326.918,Z 162.767,A -85,B 0,C 180,E1 -14932.589,E2 -14932.589} C_VEL
LIN {X 0,Y 326.753,Z 162.784,A -85,B 0,C 180,E1 -14935.065,E2 -14935.065} C_VEL
LIN {X 0,Y 326.831,Z 162.925,A -85,B 0,C 180,E1 -14936.687,E2 -14936.687} C_VEL
LIN {X 0,Y 328.109,Z 166.656,A -85,B 0,C 180,E1 -14938.159,E2 -14938.159} C_VEL
LIN {X 0,Y 329.985,Z 173.749,A -85,B 0,C 180,E1 -14940.692,E2 -14940.692} C_VEL
LIN {X 0,Y 336.004,Z 185.943,A -85,B 0,C 180,E1 -14941.892,E2 -14941.892} C_VEL
LIN {X 0,Y 340.838,Z 196.758,A -85,B 0,C 180,E1 -14942.817,E2 -14942.817} C_VEL
LIN {X 0,Y 342.431,Z 205.092,A -85,B 0,C 180,E1 -14943.267,E2 -14943.267} C_VEL
LIN {X 0,Y 338.941,Z 282.572,A -85,B 0,C 180,E1 -14945.383,E2 -14945.383} C_VEL
LIN {X 0,Y 338.026,Z 295.52,A -85,B 0,C 180,E1 -14945.967,E2 -14945.967} C_VEL
LIN {X 0,Y 336.926,Z 307.552,A -85,B 0,C 180,E1 -14946.739,E2 -14946.739} C_VEL
LIN {X 0,Y 335.455,Z 320.226,A -85,B 0,C 180,E1 -14947.827,E2 -14947.827} C_VEL
LIN {X 0,Y 333.824,Z 331.773,A -85,B 0,C 180,E1 -14949.098,E2 -14949.098} C_VEL
LIN {X 0,Y 332.065,Z 342.938,A -85,B 0,C 180,E1 -14950.673,E2 -14950.673} C_VEL
LIN {X 0,Y 330.47,Z 352.122,A -85,B 0,C 180,E1 -14952.279,E2 -14952.279} C_VEL
LIN {X 0,Y 328.889,Z 360.942,A -85,B 0,C 180,E1 -14954.226,E2 -14954.226} C_VEL
LIN {X 0,Y 327.608,Z 367.986,A -85,B 0,C 180,E1 -14956.194,E2 -14956.194} C_VEL
LIN {X 0,Y 326.61,Z 373.288,A -85,B 0,C 180,E1 -14958.089,E2 -14958.089} C_VEL
LIN {X 0,Y 325.876,Z 377.683,A -85,B 0,C 180,E1 -14960.186,E2 -14960.186} C_VEL
LIN {X 0,Y 325.413,Z 380.144,A -85,B 0,C 180,E1 -14961.768,E2 -14961.768} C_VEL
LIN {X 0,Y 325.157,Z 381.442,A -85,B 0,C 180,E1 -14962.896,E2 -14962.896} C_VEL
LIN {X 0,Y 324.886,Z 382.798,A -85,B 0,C 180,E1 -14964.692,E2 -14964.692} C_VEL
LIN {X 0,Y 324.643,Z 383.225,A -85,B 0,C 180,E1 -14967.041,E2 -14967.041} C_VEL
LIN {X 0,Y 324.633,Z 382.783,A -85,B 0,C 180,E1 -14968.443,E2 -14968.443} C_VEL
LIN {X 0,Y 324.657,Z 381.635,A -85,B 0,C 180,E1 -14970.013,E2 -14970.013} C_VEL
LIN {X 0,Y 324.745,Z 380.205,A -85,B 0,C 180,E1 -14971.292,E2 -14971.292} C_VEL
LIN {X 0,Y 325.064,Z 376.706,A -85,B 0,C 180,E1 -14973.458,E2 -14973.458} C_VEL
LIN {X 0,Y 325.389,Z 371.541,A -85,B 0,C 180,E1 -14975.674,E2 -14975.674} C_VEL
LIN {X 0,Y 325.891,Z 365.874,A -85,B 0,C 180,E1 -14977.534,E2 -14977.534} C_VEL
LIN {X 0,Y 326.482,Z 359.58,A -85,B 0,C 180,E1 -14979.198,E2 -14979.198} C_VEL
LIN {X 0,Y 327.232,Z 351.596,A -85,B 0,C 180,E1 -14980.924,E2 -14980.924} C_VEL
LIN {X 0,Y 328.05,Z 342.971,A -85,B 0,C 180,E1 -14982.443,E2 -14982.443} C_VEL
LIN {X 0,Y 329.058,Z 332.053,A -85,B 0,C 180,E1 -14983.996,E2 -14983.996} C_VEL
LIN {X 0,Y 330.06,Z 320.949,A -85,B 0,C 180,E1 -14985.261,E2 -14985.261} C_VEL
LIN {X 0,Y 331.043,Z 309.092,A -85,B 0,C 180,E1 -14986.315,E2 -14986.315} C_VEL
LIN {X 0,Y 331.836,Z 296.28,A -85,B 0,C 180,E1 -14987.185,E2 -14987.185} C_VEL
LIN {X 0,Y 332.405,Z 283.805,A -85,B 0,C 180,E1 -14987.789,E2 -14987.789} C_VEL
LIN {X 0,Y 332.938,Z 266.156,A -85,B 0,C 180,E1 -14988.309,E2 -14988.309} C_VEL
LIN {X 0,Y 334.673,Z 200.304,A -85,B 0,C 180,E1 -14989.989,E2 -14989.989} C_VEL
LIN {X 0,Y 331.225,Z 181.017,A -85,B 0,C 180,E1 -14990.696,E2 -14990.696} C_VEL
LIN {X 0,Y 328.436,Z 171.958,A -85,B 0,C 180,E1 -14991.103,E2 -14991.103} C_VEL
LIN {X 0,Y 326.694,Z 162.791,A -85,B 0,C 180,E1 -14993.92,E2 -14993.92} C_VEL
LIN {X 0,Y 326.613,Z 162.797,A -85,B 0,C 180,E1 -14997.455,E2 -14997.455} C_VEL
LIN {X 0,Y 326.585,Z 162.806,A -85,B 0,C 180,E1 -15000.332,E2 -15000.332} C_VEL
LIN {X 0,Y 326.6,Z 162.799,A -85,B 0,C 180,E1 -15003.134,E2 -15003.134} C_VEL
LIN {X 0,Y 326.596,Z 162.8,A -85,B 0,C 180,E1 -15007.21,E2 -15007.21} C_VEL
LIN {X 0,Y 326.652,Z 162.793,A -85,B 0,C 180,E1 -15011.206,E2 -15011.206} C_VEL
LIN {X 0,Y 326.73,Z 162.784,A -85,B 0,C 180,E1 -15015.458,E2 -15015.458} C_VEL
LIN {X 0,Y 326.76,Z 162.779,A -85,B 0,C 180,E1 -15018.838,E2 -15018.838} C_VEL
LIN {X 0,Y 326.917,Z 162.76,A -85,B 0,C 180,E1 -15022.588,E2 -15022.588} C_VEL
LIN {X 0,Y 326.748,Z 162.781,A -85,B 0,C 180,E1 -15025.063,E2 -15025.063} C_VEL
LIN {X 0,Y 327.012,Z 162.751,A -85,B 0,C 180,E1 -15027.535,E2 -15027.535} C_VEL
LIN {X 0,Y 327.032,Z 162.746,A -85,B 0,C 180,E1 -15031.23,E2 -15031.23} C_VEL
LIN {X 0,Y 326.752,Z 162.786,A -85,B 0,C 180,E1 -15033.699,E2 -15033.699} C_VEL
LIN {X 0,Y 326.942,Z 162.758,A -85,B 0,C 180,E1 -15036.169,E2 -15036.169} C_VEL
LIN {X 0,Y 326.784,Z 162.779,A -85,B 0,C 180,E1 -15039.906,E2 -15039.906} C_VEL
LIN {X 0,Y 326.744,Z 162.785,A -85,B 0,C 180,E1 -15043.685,E2 -15043.685} C_VEL
LIN {X 0,Y 326.629,Z 162.801,A -85,B 0,C 180,E1 -15047.531,E2 -15047.531} C_VEL
LIN {X 0,Y 326.603,Z 162.804,A -85,B 0,C 180,E1 -15051.456,E2 -15051.456} C_VEL
LIN {X 0,Y 326.6,Z 162.803,A -85,B 0,C 180,E1 -15055.49,E2 -15055.49} C_VEL
LIN {X 0,Y 326.613,Z 162.799,A -85,B 0,C 180,E1 -15059.662,E2 -15059.662} C_VEL
LIN {X 0,Y 326.616,Z 162.801,A -85,B 0,C 180,E1 -15062.945,E2 -15062.945} C_VEL
LIN {X 0,Y 326.609,Z 162.8,A -85,B 0,C 180,E1 -15065.519,E2 -15065.519} C_VEL
LIN {X 0,Y 326.587,Z 162.801,A -85,B 0,C 180,E1 -15067.677,E2 -15067.677} C_VEL
LIN {X 0,Y 325.901,Z 162.89,A -85,B 0,C 180,E1 -15068.705,E2 -15068.705} C_VEL
LIN {X 0,Y 323.086,Z 163.244,A -85,B 0,C 180,E1 -15070.381,E2 -15070.381} C_VEL
LIN {X 0,Y 320.695,Z 163.544,A -85,B 0,C 180,E1 -15071.738,E2 -15071.738} C_VEL
LIN {X 0,Y 319.638,Z 163.673,A -85,B 0,C 180,E1 -15072.788,E2 -15072.788} C_VEL
LIN {X 0,Y 319.535,Z 163.683,A -85,B 0,C 180,E1 -15073.144,E2 -15073.144} C_VEL
LIN {X 0,Y 319.547,Z 163.682,A -85,B 0,C 180,E1 -15077.015,E2 -15077.015} C_VEL
LIN {X 0,Y 319.541,Z 163.681,A -85,B 0,C 180,E1 -15080.369,E2 -15080.369} C_VEL
LIN {X 0,Y 319.575,Z 163.678,A -85,B 0,C 180,E1 -15084.456,E2 -15084.456} C_VEL
LIN {X 0,Y 319.519,Z 163.683,A -85,B 0,C 180,E1 -15088.136,E2 -15088.136} C_VEL
LIN {X 0,Y 319.564,Z 163.676,A -85,B 0,C 180,E1 -15091.603,E2 -15091.603} C_VEL
LIN {X 0,Y 319.519,Z 163.681,A -85,B 0,C 180,E1 -15095.296,E2 -15095.296} C_VEL
LIN {X 0,Y 319.556,Z 163.679,A -85,B 0,C 180,E1 -15098.044,E2 -15098.044} C_VEL
LIN {X 0,Y 319.58,Z 163.677,A -85,B 0,C 180,E1 -15102.068,E2 -15102.068} C_VEL
LIN {X 0,Y 319.702,Z 163.662,A -85,B 0,C 180,E1 -15106.006,E2 -15106.006} C_VEL
LIN {X 0,Y 319.727,Z 163.658,A -85,B 0,C 180,E1 -15109.872,E2 -15109.872} C_VEL
LIN {X 0,Y 319.892,Z 163.637,A -85,B 0,C 180,E1 -15113.693,E2 -15113.693} C_VEL
LIN {X 0,Y 319.947,Z 163.629,A -85,B 0,C 180,E1 -15117.482,E2 -15117.482} C_VEL
LIN {X 0,Y 319.99,Z 163.623,A -85,B 0,C 180,E1 -15121.258,E2 -15121.258} C_VEL
LIN {X 0,Y 319.692,Z 163.665,A -85,B 0,C 180,E1 -15123.781,E2 -15123.781} C_VEL
LIN {X 0,Y 319.891,Z 163.636,A -85,B 0,C 180,E1 -15126.306,E2 -15126.306} C_VEL
LIN {X 0,Y 319.726,Z 163.657,A -85,B 0,C 180,E1 -15130.128,E2 -15130.128} C_VEL
LIN {X 0,Y 319.701,Z 163.661,A -85,B 0,C 180,E1 -15133.993,E2 -15133.993} C_VEL
LIN {X 0,Y 319.57,Z 163.677,A -85,B 0,C 180,E1 -15137.932,E2 -15137.932} C_VEL
LIN {X 0,Y 319.552,Z 163.679,A -85,B 0,C 180,E1 -15141.955,E2 -15141.955} C_VEL
LIN {X 0,Y 319.542,Z 163.679,A -85,B 0,C 180,E1 -15146.096,E2 -15146.096} C_VEL
LIN {X 0,Y 319.533,Z 163.682,A -85,B 0,C 180,E1 -15148.939,E2 -15148.939} C_VEL
LIN {X 0,Y 319.517,Z 163.683,A -85,B 0,C 180,E1 -15151.863,E2 -15151.863} C_VEL
LIN {X 0,Y 319.572,Z 163.677,A -85,B 0,C 180,E1 -15155.543,E2 -15155.543} C_VEL
LIN {X 0,Y 319.522,Z 163.682,A -85,B 0,C 180,E1 -15159.663,E2 -15159.663} C_VEL
LIN {X 0,Y 319.512,Z 163.684,A -85,B 0,C 180,E1 -15163.461,E2 -15163.461} C_VEL
LIN {X 0,Y 319.545,Z 163.683,A -85,B 0,C 180,E1 -15167.017,E2 -15167.017} C_VEL
LIN {X 0,Y 319.54,Z 163.68,A -85,B 0,C 180,E1 -15170.371,E2 -15170.371} C_VEL
LIN {X 0,Y 319.574,Z 163.677,A -85,B 0,C 180,E1 -15174.459,E2 -15174.459} C_VEL
LIN {X 0,Y 319.52,Z 163.682,A -85,B 0,C 180,E1 -15178.138,E2 -15178.138} C_VEL
LIN {X 0,Y 319.612,Z 163.878,A -85,B 0,C 180,E1 -15179.484,E2 -15179.484} C_VEL
LIN {X 0,Y 322.289,Z 177.393,A -85,B 0,C 180,E1 -15183.389,E2 -15183.389} C_VEL
LIN {X 0,Y 323.163,Z 182.849,A -85,B 0,C 180,E1 -15184.909,E2 -15184.909} C_VEL
LIN {X 0,Y 322.548,Z 189.268,A -85,B 0,C 180,E1 -15186.587,E2 -15186.587} C_VEL
LIN {X 0,Y 327.466,Z 226.049,A -85,B 0,C 180,E1 -15187.887,E2 -15187.887} C_VEL
LIN {X 0,Y 325.555,Z 297.826,A -85,B 0,C 180,E1 -15189.795,E2 -15189.795} C_VEL
LIN {X 0,Y 324.846,Z 311.618,A -85,B 0,C 180,E1 -15190.408,E2 -15190.408} C_VEL
LIN {X 0,Y 323.994,Z 323.675,A -85,B 0,C 180,E1 -15191.177,E2 -15191.177} C_VEL
LIN {X 0,Y 322.944,Z 336.279,A -85,B 0,C 180,E1 -15192.263,E2 -15192.263} C_VEL
LIN {X 0,Y 321.831,Z 347.596,A -85,B 0,C 180,E1 -15193.509,E2 -15193.509} C_VEL
LIN {X 0,Y 320.896,Z 357.848,A -85,B 0,C 180,E1 -15194.927,E2 -15194.927} C_VEL
LIN {X 0,Y 319.902,Z 367.942,A -85,B 0,C 180,E1 -15196.664,E2 -15196.664} C_VEL
LIN {X 0,Y 319.102,Z 375.432,A -85,B 0,C 180,E1 -15198.246,E2 -15198.246} C_VEL
LIN {X 0,Y 318.501,Z 382.784,A -85,B 0,C 180,E1 -15200.155,E2 -15200.155} C_VEL
LIN {X 0,Y 318.173,Z 387.734,A -85,B 0,C 180,E1 -15201.746,E2 -15201.746} C_VEL
LIN {X 0,Y 317.912,Z 392.49,A -85,B 0,C 180,E1 -15203.655,E2 -15203.655} C_VEL
LIN {X 0,Y 317.804,Z 396.067,A -85,B 0,C 180,E1 -15205.562,E2 -15205.562} C_VEL
LIN {X 0,Y 317.769,Z 398.573,A -85,B 0,C 180,E1 -15207.466,E2 -15207.466} C_VEL
LIN {X 0,Y 317.751,Z 399.67,A -85,B 0,C 180,E1 -15208.734,E2 -15208.734} C_VEL
LIN {X 0,Y 317.785,Z 400.339,A -85,B 0,C 180,E1 -15210.001,E2 -15210.001} C_VEL
LIN {X 0,Y 317.733,Z 400.594,A -85,B 0,C 180,E1 -15211.269,E2 -15211.269} C_VEL
LIN {X 0,Y 317.754,Z 400.435,A -85,B 0,C 180,E1 -15212.536,E2 -15212.536} C_VEL
LIN {X 0,Y 317.783,Z 399.819,A -85,B 0,C 180,E1 -15213.805,E2 -15213.805} C_VEL
LIN {X 0,Y 317.825,Z 398.173,A -85,B 0,C 180,E1 -15215.687,E2 -15215.687} C_VEL
LIN {X 0,Y 318.273,Z 394.374,A -85,B 0,C 180,E1 -15218.253,E2 -15218.253} C_VEL
LIN {X 0,Y 318.851,Z 390.327,A -85,B 0,C 180,E1 -15220.157,E2 -15220.157} C_VEL
LIN {X 0,Y 319.843,Z 384.137,A -85,B 0,C 180,E1 -15222.372,E2 -15222.372} C_VEL
LIN {X 0,Y 321.183,Z 377.351,A -85,B 0,C 180,E1 -15224.252,E2 -15224.252} C_VEL
LIN {X 0,Y 322.712,Z 369.02,A -85,B 0,C 180,E1 -15226.122,E2 -15226.122} C_VEL
LIN {X 0,Y 324.073,Z 360.566,A -85,B 0,C 180,E1 -15227.676,E2 -15227.676} C_VEL
LIN {X 0,Y 325.953,Z 350.191,A -85,B 0,C 180,E1 -15229.198,E2 -15229.198} C_VEL
LIN {X 0,Y 327.846,Z 338.621,A -85,B 0,C 180,E1 -15230.551,E2 -15230.551} C_VEL
LIN {X 0,Y 329.405,Z 327.354,A -85,B 0,C 180,E1 -15231.596,E2 -15231.596} C_VEL
LIN {X 0,Y 330.718,Z 316.021,A -85,B 0,C 180,E1 -15232.408,E2 -15232.408} C_VEL
LIN {X 0,Y 332.108,Z 302.765,A -85,B 0,C 180,E1 -15233.09,E2 -15233.09} C_VEL
LIN {X 0,Y 332.908,Z 289.211,A -85,B 0,C 180,E1 -15233.566,E2 -15233.566} C_VEL
LIN {X 0,Y 335.478,Z 228.587,A -85,B 0,C 180,E1 -15235.252,E2 -15235.252} C_VEL
LIN {X 0,Y 333.182,Z 213.221,A -85,B 0,C 180,E1 -15236.036,E2 -15236.036} C_VEL
LIN {X 0,Y 329.666,Z 196.562,A -85,B 0,C 180,E1 -15237.052,E2 -15237.052} C_VEL
LIN {X 0,Y 326.538,Z 189.597,A -85,B 0,C 180,E1 -15237.715,E2 -15237.715} C_VEL
LIN {X 0,Y 325.247,Z 186.438,A -85,B 0,C 180,E1 -15238.049,E2 -15238.049} C_VEL
LIN {X 0,Y 323.636,Z 178.489,A -85,B 0,C 180,E1 -15240.686,E2 -15240.686} C_VEL
LIN {X 0,Y 321.362,Z 169.986,A -85,B 0,C 180,E1 -15243.795,E2 -15243.795} C_VEL
LIN {X 0,Y 319.557,Z 163.681,A -85,B 0,C 180,E1 -15246.366,E2 -15246.366} C_VEL
LIN {X 0,Y 319.531,Z 163.684,A -85,B 0,C 180,E1 -15249.663,E2 -15249.663} C_VEL
LIN {X 0,Y 319.522,Z 163.68,A -85,B 0,C 180,E1 -15253.461,E2 -15253.461} C_VEL
LIN {X 0,Y 319.554,Z 163.672,A -85,B 0,C 180,E1 -15257.017,E2 -15257.017} C_VEL
LIN {X 0,Y 319.517,Z 163.682,A -85,B 0,C 180,E1 -15260.367,E2 -15260.367} C_VEL
LIN {X 0,Y 319.581,Z 163.672,A -85,B 0,C 180,E1 -15264.458,E2 -15264.458} C_VEL
LIN {X 0,Y 319.527,Z 163.685,A -85,B 0,C 180,E1 -15268.138,E2 -15268.138} C_VEL
LIN {X 0,Y 319.572,Z 163.672,A -85,B 0,C 180,E1 -15271.605,E2 -15271.605} C_VEL
LIN {X 0,Y 319.544,Z 163.679,A -85,B 0,C 180,E1 -15275.299,E2 -15275.299} C_VEL
LIN {X 0,Y 319.567,Z 163.678,A -85,B 0,C 180,E1 -15278.046,E2 -15278.046} C_VEL
LIN {X 0,Y 319.591,Z 163.673,A -85,B 0,C 180,E1 -15282.069,E2 -15282.069} C_VEL
LIN {X 0,Y 319.714,Z 163.659,A -85,B 0,C 180,E1 -15286.007,E2 -15286.007} C_VEL
LIN {X 0,Y 319.74,Z 163.658,A -85,B 0,C 180,E1 -15289.873,E2 -15289.873} C_VEL
LIN {X 0,Y 319.904,Z 163.638,A -85,B 0,C 180,E1 -15293.694,E2 -15293.694} C_VEL
LIN {X 0,Y 319.739,Z 163.815,A -85,B 0,C 180,E1 -15295.667,E2 -15295.667} C_VEL
LIN {X 0,Y 321.737,Z 169.756,A -85,B 0,C 180,E1 -15298.123,E2 -15298.123} C_VEL
LIN {X 0,Y 322.924,Z 174.159,A -85,B 0,C 180,E1 -15299.721,E2 -15299.721} C_VEL
LIN {X 0,Y 329.19,Z 186.137,A -85,B 0,C 180,E1 -15301.03,E2 -15301.03} C_VEL
LIN {X 0,Y 335.115,Z 199.418,A -85,B 0,C 180,E1 -15302.241,E2 -15302.241} C_VEL
LIN {X 0,Y 336.48,Z 206.498,A -85,B 0,C 180,E1 -15302.637,E2 -15302.637} C_VEL
LIN {X 0,Y 332.827,Z 282.704,A -85,B 0,C 180,E1 -15304.772,E2 -15304.772} C_VEL
LIN {X 0,Y 331.826,Z 295.841,A -85,B 0,C 180,E1 -15305.379,E2 -15305.379} C_VEL
LIN {X 0,Y 330.53,Z 308.98,A -85,B 0,C 180,E1 -15306.256,E2 -15306.256} C_VEL
LIN {X 0,Y 329.007,Z 321.421,A -85,B 0,C 180,E1 -15307.364,E2 -15307.364} C_VEL
LIN {X 0,Y 327.297,Z 332.664,A -85,B 0,C 180,E1 -15308.645,E2 -15308.645} C_VEL
LIN {X 0,Y 325.428,Z 343.828,A -85,B 0,C 180,E1 -15310.263,E2 -15310.263} C_VEL
LIN {X 0,Y 323.691,Z 353.207,A -85,B 0,C 180,E1 -15311.974,E2 -15311.974} C_VEL
LIN {X 0,Y 322.067,Z 361.557,A -85,B 0,C 180,E1 -15313.889,E2 -15313.889} C_VEL
LIN {X 0,Y 320.667,Z 368.721,A -85,B 0,C 180,E1 -15315.968,E2 -15315.968} C_VEL
LIN {X 0,Y 319.616,Z 373.954,A -85,B 0,C 180,E1 -15317.93,E2 -15317.93} C_VEL
LIN {X 0,Y 318.868,Z 378.074,A -85,B 0,C 180,E1 -15319.976,E2 -15319.976} C_VEL
LIN {X 0,Y 318.272,Z 381.013,A -85,B 0,C 180,E1 -15322.049,E2 -15322.049} C_VEL
LIN {X 0,Y 317.975,Z 382.357,A -85,B 0,C 180,E1 -15323.444,E2 -15323.444} C_VEL
LIN {X 0,Y 317.745,Z 383.182,A -85,B 0,C 180,E1 -15324.924,E2 -15324.924} C_VEL
LIN {X 0,Y 317.588,Z 383.466,A -85,B 0,C 180,E1 -15326.269,E2 -15326.269} C_VEL
LIN {X 0,Y 317.531,Z 383.251,A -85,B 0,C 180,E1 -15327.706,E2 -15327.706} C_VEL
LIN {X 0,Y 317.527,Z 382.483,A -85,B 0,C 180,E1 -15329.14,E2 -15329.14} C_VEL
LIN {X 0,Y 317.589,Z 381.183,A -85,B 0,C 180,E1 -15330.596,E2 -15330.596} C_VEL
LIN {X 0,Y 317.875,Z 377.98,A -85,B 0,C 180,E1 -15332.842,E2 -15332.842} C_VEL
LIN {X 0,Y 318.19,Z 373.414,A -85,B 0,C 180,E1 -15335.049,E2 -15335.049} C_VEL
LIN {X 0,Y 318.663,Z 368.011,A -85,B 0,C 180,E1 -15337.013,E2 -15337.013} C_VEL
LIN {X 0,Y 319.265,Z 361.58,A -85,B 0,C 180,E1 -15338.857,E2 -15338.857} C_VEL
LIN {X 0,Y 320.06,Z 353.146,A -85,B 0,C 180,E1 -15340.788,E2 -15340.788} C_VEL
LIN {X 0,Y 320.961,Z 344.026,A -85,B 0,C 180,E1 -15342.477,E2 -15342.477} C_VEL
LIN {X 0,Y 321.938,Z 333.483,A -85,B 0,C 180,E1 -15344.042,E2 -15344.042} C_VEL
LIN {X 0,Y 323.05,Z 321.683,A -85,B 0,C 180,E1 -15345.438,E2 -15345.438} C_VEL
LIN {X 0,Y 324.072,Z 309.913,A -85,B 0,C 180,E1 -15346.521,E2 -15346.521} C_VEL
LIN {X 0,Y 324.895,Z 297.02,A -85,B 0,C 180,E1 -15347.426,E2 -15347.426} C_VEL
LIN {X 0,Y 325.477,Z 284.842,A -85,B 0,C 180,E1 -15348.043,E2 -15348.043} C_VEL
LIN {X 0,Y 326.043,Z 268.896,A -85,B 0,C 180,E1 -15348.54,E2 -15348.54} C_VEL
LIN {X 0,Y 327.817,Z 200.862,A -85,B 0,C 180,E1 -15350.323,E2 -15350.323} C_VEL
LIN {X 0,Y 324.524,Z 182.734,A -85,B 0,C 180,E1 -15351.011,E2 -15351.011} C_VEL
LIN {X 0,Y 321.242,Z 172.139,A -85,B 0,C 180,E1 -15351.506,E2 -15351.506} C_VEL
LIN {X 0,Y 319.626,Z 163.672,A -85,B 0,C 180,E1 -15354.198,E2 -15354.198} C_VEL
LIN {X 0,Y 319.529,Z 163.683,A -85,B 0,C 180,E1 -15358.137,E2 -15358.137} C_VEL
LIN {X 0,Y 319.548,Z 163.678,A -85,B 0,C 180,E1 -15361.612,E2 -15361.612} C_VEL
LIN {X 0,Y 319.53,Z 163.68,A -85,B 0,C 180,E1 -15365.297,E2 -15365.297} C_VEL
LIN {X 0,Y 319.567,Z 163.679,A -85,B 0,C 180,E1 -15368.045,E2 -15368.045} C_VEL
LIN {X 0,Y 319.589,Z 163.677,A -85,B 0,C 180,E1 -15372.068,E2 -15372.068} C_VEL
LIN {X 0,Y 319.714,Z 163.662,A -85,B 0,C 180,E1 -15376.006,E2 -15376.006} C_VEL
LIN {X 0,Y 319.739,Z 163.658,A -85,B 0,C 180,E1 -15379.871,E2 -15379.871} C_VEL
LIN {X 0,Y 319.902,Z 163.637,A -85,B 0,C 180,E1 -15383.692,E2 -15383.692} C_VEL
LIN {X 0,Y 319.958,Z 163.629,A -85,B 0,C 180,E1 -15387.481,E2 -15387.481} C_VEL
LIN {X 0,Y 320.002,Z 163.622,A -85,B 0,C 180,E1 -15391.257,E2 -15391.257} C_VEL
LIN {X 0,Y 319.702,Z 163.664,A -85,B 0,C 180,E1 -15393.78,E2 -15393.78} C_VEL
LIN {X 0,Y 319.9,Z 163.635,A -85,B 0,C 180,E1 -15396.305,E2 -15396.305} C_VEL
LIN {X 0,Y 319.736,Z 163.655,A -85,B 0,C 180,E1 -15400.127,E2 -15400.127} C_VEL
LIN {X 0,Y 319.711,Z 163.659,A -85,B 0,C 180,E1 -15403.992,E2 -15403.992} C_VEL
LIN {X 0,Y 319.58,Z 163.675,A -85,B 0,C 180,E1 -15407.93,E2 -15407.93} C_VEL
LIN {X 0,Y 319.561,Z 163.677,A -85,B 0,C 180,E1 -15411.954,E2 -15411.954} C_VEL
LIN {X 0,Y 319.549,Z 163.678,A -85,B 0,C 180,E1 -15416.094,E2 -15416.094} C_VEL
LIN {X 0,Y 319.54,Z 163.682,A -85,B 0,C 180,E1 -15418.937,E2 -15418.937} C_VEL
LIN {X 0,Y 319.523,Z 163.681,A -85,B 0,C 180,E1 -15421.861,E2 -15421.861} C_VEL
LIN {X 0,Y 319.577,Z 163.676,A -85,B 0,C 180,E1 -15425.541,E2 -15425.541} C_VEL
LIN {X 0,Y 319.526,Z 163.681,A -85,B 0,C 180,E1 -15429.661,E2 -15429.661} C_VEL
LIN {X 0,Y 319.535,Z 163.683,A -85,B 0,C 180,E1 -15433.144,E2 -15433.144} C_VEL
LIN {X 0,Y 318.816,Z 163.771,A -85,B 0,C 180,E1 -15434.195,E2 -15434.195} C_VEL
LIN {X 0,Y 315.933,Z 164.128,A -85,B 0,C 180,E1 -15435.905,E2 -15435.905} C_VEL
LIN {X 0,Y 313.525,Z 164.43,A -85,B 0,C 180,E1 -15437.291,E2 -15437.291} C_VEL
LIN {X 0,Y 312.501,Z 164.557,A -85,B 0,C 180,E1 -15438.364,E2 -15438.364} C_VEL
LIN {X 0,Y 312.421,Z 164.564,A -85,B 0,C 180,E1 -15438.728,E2 -15438.728} C_VEL
LIN {X 0,Y 312.509,Z 164.559,A -85,B 0,C 180,E1 -15442.612,E2 -15442.612} C_VEL
LIN {X 0,Y 312.515,Z 164.556,A -85,B 0,C 180,E1 -15446.31,E2 -15446.31} C_VEL
LIN {X 0,Y 312.49,Z 164.56,A -85,B 0,C 180,E1 -15450.344,E2 -15450.344} C_VEL
LIN {X 0,Y 312.501,Z 164.558,A -85,B 0,C 180,E1 -15454.1,E2 -15454.1} C_VEL
LIN {X 0,Y 312.533,Z 164.551,A -85,B 0,C 180,E1 -15457.524,E2 -15457.524} C_VEL
LIN {X 0,Y 312.544,Z 164.551,A -85,B 0,C 180,E1 -15461.65,E2 -15461.65} C_VEL
LIN {X 0,Y 312.645,Z 164.538,A -85,B 0,C 180,E1 -15465.684,E2 -15465.684} C_VEL
LIN {X 0,Y 312.677,Z 164.535,A -85,B 0,C 180,E1 -15469.641,E2 -15469.641} C_VEL
LIN {X 0,Y 312.789,Z 164.523,A -85,B 0,C 180,E1 -15472.252,E2 -15472.252} C_VEL
LIN {X 0,Y 312.68,Z 164.533,A -85,B 0,C 180,E1 -15474.841,E2 -15474.841} C_VEL
LIN {X 0,Y 312.959,Z 164.499,A -85,B 0,C 180,E1 -15478.713,E2 -15478.713} C_VEL
LIN {X 0,Y 312.959,Z 164.499,A -85,B 0,C 180,E1 -15481.286,E2 -15481.286} C_VEL
LIN {X 0,Y 312.679,Z 164.534,A -85,B 0,C 180,E1 -15485.158,E2 -15485.158} C_VEL
LIN {X 0,Y 312.789,Z 164.525,A -85,B 0,C 180,E1 -15487.748,E2 -15487.748} C_VEL
LIN {X 0,Y 312.651,Z 164.542,A -85,B 0,C 180,E1 -15491.672,E2 -15491.672} C_VEL
LIN {X 0,Y 312.606,Z 164.543,A -85,B 0,C 180,E1 -15494.828,E2 -15494.828} C_VEL
LIN {X 0,Y 312.526,Z 164.555,A -85,B 0,C 180,E1 -15499.185,E2 -15499.185} C_VEL
LIN {X 0,Y 312.506,Z 164.555,A -85,B 0,C 180,E1 -15502.775,E2 -15502.775} C_VEL
LIN {X 0,Y 312.475,Z 164.559,A -85,B 0,C 180,E1 -15506.732,E2 -15506.732} C_VEL
LIN {X 0,Y 312.487,Z 164.56,A -85,B 0,C 180,E1 -15509.656,E2 -15509.656} C_VEL
LIN {X 0,Y 312.513,Z 164.556,A -85,B 0,C 180,E1 -15513.689,E2 -15513.689} C_VEL
LIN {X 0,Y 312.506,Z 164.558,A -85,B 0,C 180,E1 -15517.388,E2 -15517.388} C_VEL
LIN {X 0,Y 312.434,Z 164.566,A -85,B 0,C 180,E1 -15520.718,E2 -15520.718} C_VEL
LIN {X 0,Y 312.444,Z 164.563,A -85,B 0,C 180,E1 -15524.211,E2 -15524.211} C_VEL
LIN {X 0,Y 312.448,Z 164.562,A -85,B 0,C 180,E1 -15527.926,E2 -15527.926} C_VEL
LIN {X 0,Y 312.478,Z 164.558,A -85,B 0,C 180,E1 -15531.924,E2 -15531.924} C_VEL
LIN {X 0,Y 312.525,Z 164.553,A -85,B 0,C 180,E1 -15534.221,E2 -15534.221} C_VEL
LIN {X 0,Y 312.497,Z 164.558,A -85,B 0,C 180,E1 -15537.335,E2 -15537.335} C_VEL
LIN {X 0,Y 312.532,Z 164.702,A -85,B 0,C 180,E1 -15539.185,E2 -15539.185} C_VEL
LIN {X 0,Y 315.168,Z 178.008,A -85,B 0,C 180,E1 -15543.122,E2 -15543.122} C_VEL
LIN {X 0,Y 316.112,Z 183.4,A -85,B 0,C 180,E1 -15544.662,E2 -15544.662} C_VEL
LIN {X 0,Y 315.682,Z 189.22,A -85,B 0,C 180,E1 -15546.199,E2 -15546.199} C_VEL
LIN {X 0,Y 320.634,Z 227.364,A -85,B 0,C 180,E1 -15547.577,E2 -15547.577} C_VEL
LIN {X 0,Y 318.652,Z 298.021,A -85,B 0,C 180,E1 -15549.506,E2 -15549.506} C_VEL
LIN {X 0,Y 317.926,Z 311.671,A -85,B 0,C 180,E1 -15550.132,E2 -15550.132} C_VEL
LIN {X 0,Y 317.067,Z 323.657,A -85,B 0,C 180,E1 -15550.918,E2 -15550.918} C_VEL
LIN {X 0,Y 315.987,Z 336.217,A -85,B 0,C 180,E1 -15552.026,E2 -15552.026} C_VEL
LIN {X 0,Y 314.853,Z 347.448,A -85,B 0,C 180,E1 -15553.291,E2 -15553.291} C_VEL
LIN {X 0,Y 313.865,Z 357.74,A -85,B 0,C 180,E1 -15554.747,E2 -15554.747} C_VEL
LIN {X 0,Y 312.906,Z 366.987,A -85,B 0,C 180,E1 -15556.36,E2 -15556.36} C_VEL
LIN {X 0,Y 311.948,Z 376,A -85,B 0,C 180,E1 -15558.303,E2 -15558.303} C_VEL
LIN {X 0,Y 311.369,Z 383.169,A -85,B 0,C 180,E1 -15560.255,E2 -15560.255} C_VEL
LIN {X 0,Y 311.002,Z 388.874,A -85,B 0,C 180,E1 -15562.209,E2 -15562.209} C_VEL
LIN {X 0,Y 310.765,Z 393.596,A -85,B 0,C 180,E1 -15564.307,E2 -15564.307} C_VEL
LIN {X 0,Y 310.744,Z 396.597,A -85,B 0,C 180,E1 -15566.111,E2 -15566.111} C_VEL
LIN {X 0,Y 310.693,Z 398.209,A -85,B 0,C 180,E1 -15567.408,E2 -15567.408} C_VEL
LIN {X 0,Y 310.665,Z 399.377,A -85,B 0,C 180,E1 -15568.705,E2 -15568.705} C_VEL
LIN {X 0,Y 310.694,Z 400.081,A -85,B 0,C 180,E1 -15570.001,E2 -15570.001} C_VEL
LIN {X 0,Y 310.648,Z 400.373,A -85,B 0,C 180,E1 -15571.297,E2 -15571.297} C_VEL
LIN {X 0,Y 310.676,Z 400.26,A -85,B 0,C 180,E1 -15572.594,E2 -15572.594} C_VEL
LIN {X 0,Y 310.695,Z 399.711,A -85,B 0,C 180,E1 -15573.892,E2 -15573.892} C_VEL
LIN {X 0,Y 310.724,Z 398.326,A -85,B 0,C 180,E1 -15575.617,E2 -15575.617} C_VEL
LIN {X 0,Y 311.086,Z 395.52,A -85,B 0,C 180,E1 -15577.792,E2 -15577.792} C_VEL
LIN {X 0,Y 311.621,Z 391.907,A -85,B 0,C 180,E1 -15579.739,E2 -15579.739} C_VEL
LIN {X 0,Y 312.436,Z 387.2,A -85,B 0,C 180,E1 -15581.681,E2 -15581.681} C_VEL
LIN {X 0,Y 313.513,Z 381.267,A -85,B 0,C 180,E1 -15583.615,E2 -15583.615} C_VEL
LIN {X 0,Y 315.073,Z 373.869,A -85,B 0,C 180,E1 -15585.527,E2 -15585.527} C_VEL
LIN {X 0,Y 316.632,Z 365.124,A -85,B 0,C 180,E1 -15587.363,E2 -15587.363} C_VEL
LIN {X 0,Y 318.517,Z 355.407,A -85,B 0,C 180,E1 -15588.994,E2 -15588.994} C_VEL
LIN {X 0,Y 320.585,Z 343.816,A -85,B 0,C 180,E1 -15590.535,E2 -15590.535} C_VEL
LIN {X 0,Y 322.451,Z 332.324,A -85,B 0,C 180,E1 -15591.749,E2 -15591.749} C_VEL
LIN {X 0,Y 324.114,Z 319.327,A -85,B 0,C 180,E1 -15592.806,E2 -15592.806} C_VEL
LIN {X 0,Y 325.686,Z 306.185,A -85,B 0,C 180,E1 -15593.572,E2 -15593.572} C_VEL
LIN {X 0,Y 326.705,Z 292.142,A -85,B 0,C 180,E1 -15594.126,E2 -15594.126} C_VEL
LIN {X 0,Y 329.547,Z 229.682,A -85,B 0,C 180,E1 -15595.904,E2 -15595.904} C_VEL
LIN {X 0,Y 327.38,Z 214.774,A -85,B 0,C 180,E1 -15596.701,E2 -15596.701} C_VEL
LIN {X 0,Y 324.137,Z 199.288,A -85,B 0,C 180,E1 -15597.685,E2 -15597.685} C_VEL
LIN {X 0,Y 319.688,Z 189.729,A -85,B 0,C 180,E1 -15598.677,E2 -15598.677} C_VEL
LIN {X 0,Y 318.131,Z 186.171,A -85,B 0,C 180,E1 -15599.08,E2 -15599.08} C_VEL
LIN {X 0,Y 316.664,Z 179.403,A -85,B 0,C 180,E1 -15601.438,E2 -15601.438} C_VEL
LIN {X 0,Y 314.096,Z 169.749,A -85,B 0,C 180,E1 -15605.182,E2 -15605.182} C_VEL
LIN {X 0,Y 312.509,Z 164.555,A -85,B 0,C 180,E1 -15607.474,E2 -15607.474} C_VEL
LIN {X 0,Y 312.443,Z 164.566,A -85,B 0,C 180,E1 -15610.718,E2 -15610.718} C_VEL
LIN {X 0,Y 312.453,Z 164.561,A -85,B 0,C 180,E1 -15614.211,E2 -15614.211} C_VEL
LIN {X 0,Y 312.458,Z 164.559,A -85,B 0,C 180,E1 -15617.925,E2 -15617.925} C_VEL
LIN {X 0,Y 312.479,Z 164.555,A -85,B 0,C 180,E1 -15621.925,E2 -15621.925} C_VEL
LIN {X 0,Y 312.533,Z 164.549,A -85,B 0,C 180,E1 -15624.221,E2 -15624.221} C_VEL
LIN {X 0,Y 312.505,Z 164.557,A -85,B 0,C 180,E1 -15627.334,E2 -15627.334} C_VEL
LIN {X 0,Y 312.508,Z 164.553,A -85,B 0,C 180,E1 -15631.293,E2 -15631.293} C_VEL
LIN {X 0,Y 312.525,Z 164.55,A -85,B 0,C 180,E1 -15634.706,E2 -15634.706} C_VEL
LIN {X 0,Y 312.543,Z 164.55,A -85,B 0,C 180,E1 -15637.526,E2 -15637.526} C_VEL
LIN {X 0,Y 312.555,Z 164.548,A -85,B 0,C 180,E1 -15641.652,E2 -15641.652} C_VEL
LIN {X 0,Y 312.656,Z 164.539,A -85,B 0,C 180,E1 -15645.685,E2 -15645.685} C_VEL
LIN {X 0,Y 312.69,Z 164.537,A -85,B 0,C 180,E1 -15649.642,E2 -15649.642} C_VEL
LIN {X 0,Y 312.8,Z 164.524,A -85,B 0,C 180,E1 -15652.253,E2 -15652.253} C_VEL
LIN {X 0,Y 312.731,Z 164.607,A -85,B 0,C 180,E1 -15654.52,E2 -15654.52} C_VEL
LIN {X 0,Y 314.986,Z 171.282,A -85,B 0,C 180,E1 -15657.443,E2 -15657.443} C_VEL
LIN {X 0,Y 315.787,Z 174.503,A -85,B 0,C 180,E1 -15658.645,E2 -15658.645} C_VEL
LIN {X 0,Y 322.494,Z 186.699,A -85,B 0,C 180,E1 -15660.138,E2 -15660.138} C_VEL
LIN {X 0,Y 329.643,Z 202.507,A -85,B 0,C 180,E1 -15661.671,E2 -15661.671} C_VEL
LIN {X 0,Y 330.614,Z 207.378,A -85,B 0,C 180,E1 -15661.968,E2 -15661.968} C_VEL
LIN {X 0,Y 326.79,Z 282.811,A -85,B 0,C 180,E1 -15664.124,E2 -15664.124} C_VEL
LIN {X 0,Y 325.771,Z 295.58,A -85,B 0,C 180,E1 -15664.718,E2 -15664.718} C_VEL
LIN {X 0,Y 324.553,Z 307.561,A -85,B 0,C 180,E1 -15665.507,E2 -15665.507} C_VEL
LIN {X 0,Y 323.03,Z 319.543,A -85,B 0,C 180,E1 -15666.559,E2 -15666.559} C_VEL
LIN {X 0,Y 321.253,Z 331.022,A -85,B 0,C 180,E1 -15667.844,E2 -15667.844} C_VEL
LIN {X 0,Y 319.383,Z 341.638,A -85,B 0,C 180,E1 -15669.34,E2 -15669.34} C_VEL
LIN {X 0,Y 317.679,Z 350.278,A -85,B 0,C 180,E1 -15670.839,E2 -15670.839} C_VEL
LIN {X 0,Y 316.198,Z 357.851,A -85,B 0,C 180,E1 -15672.448,E2 -15672.448} C_VEL
LIN {X 0,Y 314.769,Z 364.676,A -85,B 0,C 180,E1 -15674.218,E2 -15674.218} C_VEL
LIN {X 0,Y 313.41,Z 371.013,A -85,B 0,C 180,E1 -15676.278,E2 -15676.278} C_VEL
LIN {X 0,Y 312.368,Z 375.925,A -85,B 0,C 180,E1 -15678.36,E2 -15678.36} C_VEL
LIN {X 0,Y 311.628,Z 379.566,A -85,B 0,C 180,E1 -15680.461,E2 -15680.461} C_VEL
LIN {X 0,Y 311.052,Z 382.055,A -85,B 0,C 180,E1 -15682.589,E2 -15682.589} C_VEL
LIN {X 0,Y 310.771,Z 383.087,A -85,B 0,C 180,E1 -15684.021,E2 -15684.021} C_VEL
LIN {X 0,Y 310.577,Z 383.619,A -85,B 0,C 180,E1 -15685.465,E2 -15685.465} C_VEL
LIN {X 0,Y 310.435,Z 383.268,A -85,B 0,C 180,E1 -15688,E2 -15688} C_VEL
LIN {X 0,Y 310.494,Z 381.189,A -85,B 0,C 180,E1 -15690.668,E2 -15690.668} C_VEL
LIN {X 0,Y 310.778,Z 378.062,A -85,B 0,C 180,E1 -15692.871,E2 -15692.871} C_VEL
LIN {X 0,Y 311.103,Z 373.756,A -85,B 0,C 180,E1 -15694.999,E2 -15694.999} C_VEL
LIN {X 0,Y 311.6,Z 368.088,A -85,B 0,C 180,E1 -15697.11,E2 -15697.11} C_VEL
LIN {X 0,Y 312.328,Z 360.259,A -85,B 0,C 180,E1 -15699.342,E2 -15699.342} C_VEL
LIN {X 0,Y 313.062,Z 352.803,A -85,B 0,C 180,E1 -15701.045,E2 -15701.045} C_VEL
LIN {X 0,Y 313.907,Z 344.513,A -85,B 0,C 180,E1 -15702.605,E2 -15702.605} C_VEL
LIN {X 0,Y 314.886,Z 334.527,A -85,B 0,C 180,E1 -15704.141,E2 -15704.141} C_VEL
LIN {X 0,Y 316.027,Z 322.643,A -85,B 0,C 180,E1 -15705.596,E2 -15705.596} C_VEL
LIN {X 0,Y 317.053,Z 311.273,A -85,B 0,C 180,E1 -15706.693,E2 -15706.693} C_VEL
LIN {X 0,Y 317.929,Z 298.04,A -85,B 0,C 180,E1 -15707.66,E2 -15707.66} C_VEL
LIN {X 0,Y 318.608,Z 284.812,A -85,B 0,C 180,E1 -15708.352,E2 -15708.352} C_VEL
LIN {X 0,Y 319.171,Z 268.154,A -85,B 0,C 180,E1 -15708.877,E2 -15708.877} C_VEL
LIN {X 0,Y 321.061,Z 202.189,A -85,B 0,C 180,E1 -15710.644,E2 -15710.644} C_VEL
LIN {X 0,Y 317.99,Z 184.931,A -85,B 0,C 180,E1 -15711.313,E2 -15711.313} C_VEL
LIN {X 0,Y 314.044,Z 172.233,A -85,B 0,C 180,E1 -15711.947,E2 -15711.947} C_VEL
LIN {X 0,Y 312.556,Z 164.554,A -85,B 0,C 180,E1 -15714.421,E2 -15714.421} C_VEL
LIN {X 0,Y 312.507,Z 164.555,A -85,B 0,C 180,E1 -15717.333,E2 -15717.333} C_VEL
LIN {X 0,Y 312.489,Z 164.557,A -85,B 0,C 180,E1 -15721.299,E2 -15721.299} C_VEL
LIN {X 0,Y 312.521,Z 164.555,A -85,B 0,C 180,E1 -15724.704,E2 -15724.704} C_VEL
LIN {X 0,Y 312.544,Z 164.551,A -85,B 0,C 180,E1 -15727.525,E2 -15727.525} C_VEL
LIN {X 0,Y 312.55,Z 164.551,A -85,B 0,C 180,E1 -15731.65,E2 -15731.65} C_VEL
LIN {X 0,Y 312.656,Z 164.538,A -85,B 0,C 180,E1 -15735.683,E2 -15735.683} C_VEL
LIN {X 0,Y 312.689,Z 164.534,A -85,B 0,C 180,E1 -15739.64,E2 -15739.64} C_VEL
LIN {X 0,Y 312.8,Z 164.521,A -85,B 0,C 180,E1 -15742.251,E2 -15742.251} C_VEL
LIN {X 0,Y 312.689,Z 164.532,A -85,B 0,C 180,E1 -15744.841,E2 -15744.841} C_VEL
LIN {X 0,Y 312.971,Z 164.497,A -85,B 0,C 180,E1 -15748.712,E2 -15748.712} C_VEL
LIN {X 0,Y 312.97,Z 164.498,A -85,B 0,C 180,E1 -15751.286,E2 -15751.286} C_VEL
LIN {X 0,Y 312.688,Z 164.533,A -85,B 0,C 180,E1 -15755.157,E2 -15755.157} C_VEL
LIN {X 0,Y 312.798,Z 164.523,A -85,B 0,C 180,E1 -15757.746,E2 -15757.746} C_VEL
LIN {X 0,Y 312.662,Z 164.54,A -85,B 0,C 180,E1 -15761.67,E2 -15761.67} C_VEL
LIN {X 0,Y 312.616,Z 164.542,A -85,B 0,C 180,E1 -15764.826,E2 -15764.826} C_VEL
LIN {X 0,Y 312.534,Z 164.555,A -85,B 0,C 180,E1 -15769.184,E2 -15769.184} C_VEL
LIN {X 0,Y 312.514,Z 164.555,A -85,B 0,C 180,E1 -15772.774,E2 -15772.774} C_VEL
LIN {X 0,Y 312.483,Z 164.559,A -85,B 0,C 180,E1 -15776.731,E2 -15776.731} C_VEL
LIN {X 0,Y 312.494,Z 164.558,A -85,B 0,C 180,E1 -15779.654,E2 -15779.654} C_VEL
LIN {X 0,Y 312.518,Z 164.554,A -85,B 0,C 180,E1 -15783.687,E2 -15783.687} C_VEL
LIN {X 0,Y 312.511,Z 164.557,A -85,B 0,C 180,E1 -15787.386,E2 -15787.386} C_VEL
LIN {X 0,Y 312.438,Z 164.566,A -85,B 0,C 180,E1 -15790.716,E2 -15790.716} C_VEL
LIN {X 0,Y 312.447,Z 164.563,A -85,B 0,C 180,E1 -15794.209,E2 -15794.209} C_VEL
LIN {X 0,Y 312.45,Z 164.562,A -85,B 0,C 180,E1 -15797.924,E2 -15797.924} C_VEL
LIN {X 0,Y 312.421,Z 164.564,A -85,B 0,C 180,E1 -15798.728,E2 -15798.728} C_VEL
LIN {X 0,Y 311.765,Z 164.648,A -85,B 0,C 180,E1 -15799.803,E2 -15799.803} C_VEL
LIN {X 0,Y 308.93,Z 165,A -85,B 0,C 180,E1 -15801.554,E2 -15801.554} C_VEL
LIN {X 0,Y 306.532,Z 165.302,A -85,B 0,C 180,E1 -15802.974,E2 -15802.974} C_VEL
LIN {X 0,Y 305.516,Z 165.426,A -85,B 0,C 180,E1 -15804.073,E2 -15804.073} C_VEL
LIN {X 0,Y 305.441,Z 165.435,A -85,B 0,C 180,E1 -15804.445,E2 -15804.445} C_VEL
LIN {X 0,Y 305.437,Z 165.438,A -85,B 0,C 180,E1 -15808.357,E2 -15808.357} C_VEL
LIN {X 0,Y 305.469,Z 165.433,A -85,B 0,C 180,E1 -15811.108,E2 -15811.108} C_VEL
